LIN {X 0,Y 308.222,Z 305.882,A -85,B 0,C 180,E1 -15823.701,E2 -15823.701} C_VEL
LIN {X 0,Y 306.915,Z 363.331,A -85,B 0,C 180,E1 -15825.712,E2 -15825.712} C_VEL
LIN {X 0,Y 306.575,Z 374.52,A -85,B 0,C 180,E1 -15826.33,E2 -15826.33} C_VEL
LIN {X 0,Y 306.13,Z 386.23,A -85,B 0,C 180,E1 -15827.239,E2 -15827.239} C_VEL
LIN {X 0,Y 305.731,Z 395.85,A -85,B 0,C 180,E1 -15828.233,E2 -15828.233} C_VEL
LIN {X 0,Y 305.222,Z 403.664,A -85,B 0,C 180,E1 -15829.222,E2 -15829.222} C_VEL
LIN {X 0,Y 304.911,Z 411.279,A -85,B 0,C 180,E1 -15830.385,E2 -15830.385} C_VEL
LIN {X 0,Y 304.492,Z 420.077,A -85,B 0,C 180,E1 -15832.044,E2 -15832.044} C_VEL
LIN {X 0,Y 304.105,Z 426.542,A -85,B 0,C 180,E1 -15833.594,E2 -15833.594} C_VEL
LIN {X 0,Y 303.997,Z 432.469,A -85,B 0,C 180,E1 -15835.363,E2 -15835.363} C_VEL
LIN {X 0,Y 303.844,Z 436.01,A -85,B 0,C 180,E1 -15836.689,E2 -15836.689} C_VEL
LIN {X 0,Y 303.696,Z 438.88,A -85,B 0,C 180,E1 -15838.015,E2 -15838.015} C_VEL
LIN {X 0,Y 303.696,Z 442.054,A -85,B 0,C 180,E1 -15840.004,E2 -15840.004} C_VEL
LIN {X 0,Y 303.79,Z 443.417,A -85,B 0,C 180,E1 -15841.33,E2 -15841.33} C_VEL
LIN {X 0,Y 303.999,Z 444.25,A -85,B 0,C 180,E1 -15842.654,E2 -15842.654} C_VEL
LIN {X 0,Y 304.362,Z 444.561,A -85,B 0,C 180,E1 -15843.976,E2 -15843.976} C_VEL
LIN {X 0,Y 304.785,Z 444.334,A -85,B 0,C 180,E1 -15845.296,E2 -15845.296} C_VEL
LIN {X 0,Y 305.137,Z 443.516,A -85,B 0,C 180,E1 -15846.617,E2 -15846.617} C_VEL
LIN {X 0,Y 305.482,Z 442.17,A -85,B 0,C 180,E1 -15847.938,E2 -15847.938} C_VEL
LIN {X 0,Y 306.786,Z 439.095,A -85,B 0,C 180,E1 -15849.913,E2 -15849.913} C_VEL
LIN {X 0,Y 308.158,Z 434.613,A -85,B 0,C 180,E1 -15851.848,E2 -15851.848} C_VEL
LIN {X 0,Y 309.858,Z 428.578,A -85,B 0,C 180,E1 -15853.781,E2 -15853.781} C_VEL
LIN {X 0,Y 311.569,Z 422.164,A -85,B 0,C 180,E1 -15855.373,E2 -15855.373} C_VEL
LIN {X 0,Y 313.433,Z 413.992,A -85,B 0,C 180,E1 -15856.951,E2 -15856.951} C_VEL
LIN {X 0,Y 315.28,Z 404.81,A -85,B 0,C 180,E1 -15858.356,E2 -15858.356} C_VEL
LIN {X 0,Y 317.115,Z 394.594,A -85,B 0,C 180,E1 -15859.589,E2 -15859.589} C_VEL
LIN {X 0,Y 318.559,Z 384.696,A -85,B 0,C 180,E1 -15860.505,E2 -15860.505} C_VEL
LIN {X 0,Y 319.952,Z 372.941,A -85,B 0,C 180,E1 -15861.338,E2 -15861.338} C_VEL
LIN {X 0,Y 321.066,Z 360.035,A -85,B 0,C 180,E1 -15861.94,E2 -15861.94} C_VEL
LIN {X 0,Y 324.472,Z 318.367,A -85,B 0,C 180,E1 -15863.552,E2 -15863.552} C_VEL
LIN {X 0,Y 320.07,Z 308.921,A -85,B 0,C 180,E1 -15864.841,E2 -15864.841} C_VEL
LIN {X 0,Y 315.605,Z 300.854,A -85,B 0,C 180,E1 -15866.21,E2 -15866.21} C_VEL
LIN {X 0,Y 313.092,Z 296.819,A -85,B 0,C 180,E1 -15867.028,E2 -15867.028} C_VEL
LIN {X 0,Y 310.13,Z 292.309,A -85,B 0,C 180,E1 -15868.032,E2 -15868.032} C_VEL
LIN {X 0,Y 307.849,Z 288.757,A -85,B 0,C 180,E1 -15868.912,E2 -15868.912} C_VEL
LIN {X 0,Y 306.286,Z 284.748,A -85,B 0,C 180,E1 -15871.087,E2 -15871.087} C_VEL
LIN {X 0,Y 305.48,Z 282.247,A -85,B 0,C 180,E1 -15872.536,E2 -15872.536} C_VEL
LIN {X 0,Y 305.461,Z 282.248,A -85,B 0,C 180,E1 -15876.745,E2 -15876.745} C_VEL
LIN {X 0,Y 305.42,Z 282.253,A -85,B 0,C 180,E1 -15880.592,E2 -15880.592} C_VEL
LIN {X 0,Y 305.432,Z 282.249,A -85,B 0,C 180,E1 -15883.658,E2 -15883.658} C_VEL
LIN {X 0,Y 305.453,Z 282.246,A -85,B 0,C 180,E1 -15887.419,E2 -15887.419} C_VEL
LIN {X 0,Y 305.469,Z 282.246,A -85,B 0,C 180,E1 -15889.894,E2 -15889.894} C_VEL
LIN {X 0,Y 305.474,Z 282.24,A -85,B 0,C 180,E1 -15893.638,E2 -15893.638} C_VEL
LIN {X 0,Y 305.483,Z 282.361,A -85,B 0,C 180,E1 -15896.831,E2 -15896.831} C_VEL
LIN {X 0,Y 306.911,Z 285.743,A -85,B 0,C 180,E1 -15898.218,E2 -15898.218} C_VEL
LIN {X 0,Y 308.188,Z 287.872,A -85,B 0,C 180,E1 -15899.13,E2 -15899.13} C_VEL
LIN {X 0,Y 311.974,Z 294.665,A -85,B 0,C 180,E1 -15901.475,E2 -15901.475} C_VEL
LIN {X 0,Y 313.574,Z 299.445,A -85,B 0,C 180,E1 -15902.559,E2 -15902.559} C_VEL
LIN {X 0,Y 316.579,Z 307.966,A -85,B 0,C 180,E1 -15903.728,E2 -15903.728} C_VEL
LIN {X 0,Y 319.09,Z 321.708,A -85,B 0,C 180,E1 -15905.03,E2 -15905.03} C_VEL
LIN {X 0,Y 321.279,Z 340.372,A -85,B 0,C 180,E1 -15906.429,E2 -15906.429} C_VEL
LIN {X 0,Y 321.899,Z 352.846,A -85,B 0,C 180,E1 -15907.185,E2 -15907.185} C_VEL
LIN {X 0,Y 318.853,Z 391.341,A -85,B 0,C 180,E1 -15908.715,E2 -15908.715} C_VEL
LIN {X 0,Y 317.251,Z 403.092,A -85,B 0,C 180,E1 -15909.41,E2 -15909.41} C_VEL
LIN {X 0,Y 315.418,Z 414.235,A -85,B 0,C 180,E1 -15910.305,E2 -15910.305} C_VEL
LIN {X 0,Y 313.271,Z 425.528,A -85,B 0,C 180,E1 -15911.525,E2 -15911.525} C_VEL
LIN {X 0,Y 311.637,Z 433.396,A -85,B 0,C 180,E1 -15912.613,E2 -15912.613} C_VEL
LIN {X 0,Y 310.356,Z 439.144,A -85,B 0,C 180,E1 -15913.557,E2 -15913.557} C_VEL
LIN {X 0,Y 308.572,Z 447.09,A -85,B 0,C 180,E1 -15915.153,E2 -15915.153} C_VEL
LIN {X 0,Y 307.019,Z 453.583,A -85,B 0,C 180,E1 -15916.767,E2 -15916.767} C_VEL
LIN {X 0,Y 305.696,Z 459.553,A -85,B 0,C 180,E1 -15918.731,E2 -15918.731} C_VEL
LIN {X 0,Y 304.665,Z 464.003,A -85,B 0,C 180,E1 -15920.707,E2 -15920.707} C_VEL
LIN {X 0,Y 304.18,Z 466.239,A -85,B 0,C 180,E1 -15922.031,E2 -15922.031} C_VEL
LIN {X 0,Y 303.857,Z 467.931,A -85,B 0,C 180,E1 -15923.359,E2 -15923.359} C_VEL
LIN {X 0,Y 303.703,Z 469.072,A -85,B 0,C 180,E1 -15924.689,E2 -15924.689} C_VEL
LIN {X 0,Y 303.705,Z 469.6,A -85,B 0,C 180,E1 -15926.019,E2 -15926.019} C_VEL
LIN {X 0,Y 303.7,Z 469.578,A -85,B 0,C 180,E1 -15927.347,E2 -15927.347} C_VEL
LIN {X 0,Y 303.732,Z 470.856,A -85,B 0,C 180,E1 -15928.674,E2 -15928.674} C_VEL
LIN {X 0,Y 303.767,Z 471.719,A -85,B 0,C 180,E1 -15930,E2 -15930} C_VEL
LIN {X 0,Y 303.675,Z 472.01,A -85,B 0,C 180,E1 -15931.326,E2 -15931.326} C_VEL
LIN {X 0,Y 303.669,Z 471.757,A -85,B 0,C 180,E1 -15932.653,E2 -15932.653} C_VEL
LIN {X 0,Y 303.693,Z 471.045,A -85,B 0,C 180,E1 -15933.981,E2 -15933.981} C_VEL
LIN {X 0,Y 303.741,Z 469.324,A -85,B 0,C 180,E1 -15935.745,E2 -15935.745} C_VEL
LIN {X 0,Y 303.981,Z 467.036,A -85,B 0,C 180,E1 -15937.305,E2 -15937.305} C_VEL
LIN {X 0,Y 304.552,Z 462.968,A -85,B 0,C 180,E1 -15939.296,E2 -15939.296} C_VEL
LIN {X 0,Y 305.469,Z 457.514,A -85,B 0,C 180,E1 -15941.277,E2 -15941.277} C_VEL
LIN {X 0,Y 306.487,Z 451.586,A -85,B 0,C 180,E1 -15942.919,E2 -15942.919} C_VEL
LIN {X 0,Y 307.726,Z 444.1,A -85,B 0,C 180,E1 -15944.55,E2 -15944.55} C_VEL
LIN {X 0,Y 309.047,Z 436.733,A -85,B 0,C 180,E1 -15945.836,E2 -15945.836} C_VEL
LIN {X 0,Y 310.236,Z 428.868,A -85,B 0,C 180,E1 -15946.957,E2 -15946.957} C_VEL
LIN {X 0,Y 311.491,Z 420.567,A -85,B 0,C 180,E1 -15947.903,E2 -15947.903} C_VEL
LIN {X 0,Y 312.707,Z 410.021,A -85,B 0,C 180,E1 -15948.849,E2 -15948.849} C_VEL
LIN {X 0,Y 313.833,Z 398.627,A -85,B 0,C 180,E1 -15949.543,E2 -15949.543} C_VEL
LIN {X 0,Y 314.465,Z 389.052,A -85,B 0,C 180,E1 -15949.934,E2 -15949.934} C_VEL
LIN {X 0,Y 315.324,Z 349.248,A -85,B 0,C 180,E1 -15950.906,E2 -15950.906} C_VEL
LIN {X 0,Y 312.484,Z 330.482,A -85,B 0,C 180,E1 -15951.629,E2 -15951.629} C_VEL
LIN {X 0,Y 308.344,Z 310.347,A -85,B 0,C 180,E1 -15952.538,E2 -15952.538} C_VEL
LIN {X 0,Y 309.432,Z 302.136,A -85,B 0,C 180,E1 -15954.993,E2 -15954.993} C_VEL
LIN {X 0,Y 308.381,Z 295.263,A -85,B 0,C 180,E1 -15957.271,E2 -15957.271} C_VEL
LIN {X 0,Y 306.222,Z 285.499,A -85,B 0,C 180,E1 -15960.707,E2 -15960.707} C_VEL
LIN {X 0,Y 305.446,Z 282.244,A -85,B 0,C 180,E1 -15961.952,E2 -15961.952} C_VEL
LIN {X 0,Y 305.47,Z 282.239,A -85,B 0,C 180,E1 -15965.112,E2 -15965.112} C_VEL
LIN {X 0,Y 305.436,Z 282.251,A -85,B 0,C 180,E1 -15968.521,E2 -15968.521} C_VEL
LIN {X 0,Y 305.449,Z 282.248,A -85,B 0,C 180,E1 -15971.855,E2 -15971.855} C_VEL
LIN {X 0,Y 305.409,Z 282.255,A -85,B 0,C 180,E1 -15975.509,E2 -15975.509} C_VEL
LIN {X 0,Y 305.421,Z 282.251,A -85,B 0,C 180,E1 -15978.136,E2 -15978.136} C_VEL
LIN {X 0,Y 305.45,Z 282.244,A -85,B 0,C 180,E1 -15981.59,E2 -15981.59} C_VEL
LIN {X 0,Y 305.47,Z 282.238,A -85,B 0,C 180,E1 -15984.884,E2 -15984.884} C_VEL
LIN {X 0,Y 305.449,Z 282.242,A -85,B 0,C 180,E1 -15988.356,E2 -15988.356} C_VEL
LIN {X 0,Y 305.493,Z 282.242,A -85,B 0,C 180,E1 -15991.107,E2 -15991.107} C_VEL
LIN {X 0,Y 305.51,Z 282.235,A -85,B 0,C 180,E1 -15994.079,E2 -15994.079} C_VEL
LIN {X 0,Y 305.481,Z 282.234,A -85,B 0,C 180,E1 -15998.398,E2 -15998.398} C_VEL
LIN {X 0,Y 305.548,Z 282.235,A -85,B 0,C 180,E1 -16001.211,E2 -16001.211} C_VEL
LIN {X 0,Y 305.631,Z 282.22,A -85,B 0,C 180,E1 -16005.344,E2 -16005.344} C_VEL
LIN {X 0,Y 305.639,Z 282.21,A -85,B 0,C 180,E1 -16009.396,E2 -16009.396} C_VEL
LIN {X 0,Y 305.8,Z 282.202,A -85,B 0,C 180,E1 -16012.07,E2 -16012.07} C_VEL
LIN {X 0,Y 305.681,Z 282.205,A -85,B 0,C 180,E1 -16014.719,E2 -16014.719} C_VEL
LIN {X 0,Y 305.952,Z 282.176,A -85,B 0,C 180,E1 -16018.68,E2 -16018.68} C_VEL
LIN {X 0,Y 305.951,Z 282.178,A -85,B 0,C 180,E1 -16021.312,E2 -16021.312} C_VEL
LIN {X 0,Y 305.669,Z 282.207,A -85,B 0,C 180,E1 -16025.272,E2 -16025.272} C_VEL
LIN {X 0,Y 305.76,Z 282.209,A -85,B 0,C 180,E1 -16027.922,E2 -16027.922} C_VEL
LIN {X 0,Y 305.594,Z 282.225,A -85,B 0,C 180,E1 -16031.941,E2 -16031.941} C_VEL
LIN {X 0,Y 305.631,Z 282.218,A -85,B 0,C 180,E1 -16035.03,E2 -16035.03} C_VEL
LIN {X 0,Y 305.568,Z 282.23,A -85,B 0,C 180,E1 -16039.44,E2 -16039.44} C_VEL
LIN {X 0,Y 305.48,Z 282.244,A -85,B 0,C 180,E1 -16043.037,E2 -16043.037} C_VEL
LIN {X 0,Y 305.534,Z 282.238,A -85,B 0,C 180,E1 -16046.222,E2 -16046.222} C_VEL
LIN {X 0,Y 305.474,Z 282.244,A -85,B 0,C 180,E1 -16049.043,E2 -16049.043} C_VEL
LIN {X 0,Y 305.426,Z 282.248,A -85,B 0,C 180,E1 -16051.948,E2 -16051.948} C_VEL
LIN {X 0,Y 305.445,Z 282.237,A -85,B 0,C 180,E1 -16055.109,E2 -16055.109} C_VEL
LIN {X 0,Y 305.464,Z 282.25,A -85,B 0,C 180,E1 -16058.532,E2 -16058.532} C_VEL
LIN {X 0,Y 305.5,Z 282.247,A -85,B 0,C 180,E1 -16062.595,E2 -16062.595} C_VEL
LIN {X 0,Y 305.511,Z 282.24,A -85,B 0,C 180,E1 -16066.36,E2 -16066.36} C_VEL
LIN {X 0,Y 305.504,Z 282.301,A -85,B 0,C 180,E1 -16069.07,E2 -16069.07} C_VEL
LIN {X 0,Y 306.197,Z 285.476,A -85,B 0,C 180,E1 -16070.276,E2 -16070.276} C_VEL
LIN {X 0,Y 314.034,Z 303.632,A -85,B 0,C 180,E1 -16071.501,E2 -16071.501} C_VEL
LIN {X 0,Y 315.844,Z 309.078,A -85,B 0,C 180,E1 -16071.805,E2 -16071.805} C_VEL
LIN {X 0,Y 316.318,Z 312.256,A -85,B 0,C 180,E1 -16071.928,E2 -16071.928} C_VEL
LIN {X 0,Y 315.025,Z 362.447,A -85,B 0,C 180,E1 -16073.124,E2 -16073.124} C_VEL
LIN {X 0,Y 314.521,Z 372.658,A -85,B 0,C 180,E1 -16073.558,E2 -16073.558} C_VEL
LIN {X 0,Y 313.622,Z 384.807,A -85,B 0,C 180,E1 -16074.364,E2 -16074.364} C_VEL
LIN {X 0,Y 312.594,Z 394.073,A -85,B 0,C 180,E1 -16075.215,E2 -16075.215} C_VEL
LIN {X 0,Y 311.639,Z 402.117,A -85,B 0,C 180,E1 -16076.158,E2 -16076.158} C_VEL
LIN {X 0,Y 310.511,Z 409.965,A -85,B 0,C 180,E1 -16077.291,E2 -16077.291} C_VEL
LIN {X 0,Y 309.347,Z 416.815,A -85,B 0,C 180,E1 -16078.498,E2 -16078.498} C_VEL
LIN {X 0,Y 308.024,Z 424.176,A -85,B 0,C 180,E1 -16080.102,E2 -16080.102} C_VEL
LIN {X 0,Y 306.792,Z 430.833,A -85,B 0,C 180,E1 -16081.991,E2 -16081.991} C_VEL
LIN {X 0,Y 305.862,Z 435.31,A -85,B 0,C 180,E1 -16083.64,E2 -16083.64} C_VEL
LIN {X 0,Y 305.059,Z 439.119,A -85,B 0,C 180,E1 -16085.501,E2 -16085.501} C_VEL
LIN {X 0,Y 304.433,Z 441.868,A -85,B 0,C 180,E1 -16087.415,E2 -16087.415} C_VEL
LIN {X 0,Y 304.202,Z 442.815,A -85,B 0,C 180,E1 -16088.306,E2 -16088.306} C_VEL
LIN {X 0,Y 303.9,Z 443.783,A -85,B 0,C 180,E1 -16089.703,E2 -16089.703} C_VEL
LIN {X 0,Y 303.654,Z 444.181,A -85,B 0,C 180,E1 -16091.591,E2 -16091.591} C_VEL
LIN {X 0,Y 303.571,Z 443.264,A -85,B 0,C 180,E1 -16093.871,E2 -16093.871} C_VEL
LIN {X 0,Y 303.662,Z 442.055,A -85,B 0,C 180,E1 -16095.251,E2 -16095.251} C_VEL
LIN {X 0,Y 303.816,Z 440.306,A -85,B 0,C 180,E1 -16096.625,E2 -16096.625} C_VEL
LIN {X 0,Y 304.15,Z 436.443,A -85,B 0,C 180,E1 -16098.673,E2 -16098.673} C_VEL
LIN {X 0,Y 304.596,Z 431.173,A -85,B 0,C 180,E1 -16100.706,E2 -16100.706} C_VEL
LIN {X 0,Y 305.064,Z 425.345,A -85,B 0,C 180,E1 -16102.436,E2 -16102.436} C_VEL
LIN {X 0,Y 305.742,Z 418.331,A -85,B 0,C 180,E1 -16104.063,E2 -16104.063} C_VEL
LIN {X 0,Y 306.469,Z 410.103,A -85,B 0,C 180,E1 -16105.561,E2 -16105.561} C_VEL
LIN {X 0,Y 307.174,Z 402.221,A -85,B 0,C 180,E1 -16106.721,E2 -16106.721} C_VEL
LIN {X 0,Y 307.818,Z 393.913,A -85,B 0,C 180,E1 -16107.71,E2 -16107.71} C_VEL
LIN {X 0,Y 308.409,Z 385.228,A -85,B 0,C 180,E1 -16108.531,E2 -16108.531} C_VEL
LIN {X 0,Y 309,Z 373.68,A -85,B 0,C 180,E1 -16109.349,E2 -16109.349} C_VEL
LIN {X 0,Y 309.302,Z 362.42,A -85,B 0,C 180,E1 -16109.854,E2 -16109.854} C_VEL
LIN {X 0,Y 309.849,Z 331.975,A -85,B 0,C 180,E1 -16110.602,E2 -16110.602} C_VEL
LIN {X 0,Y 310.282,Z 307.413,A -85,B 0,C 180,E1 -16111.166,E2 -16111.166} C_VEL
LIN {X 0,Y 306.839,Z 286.854,A -85,B 0,C 180,E1 -16111.821,E2 -16111.821} C_VEL
LIN {X 0,Y 306.326,Z 284.637,A -85,B 0,C 180,E1 -16111.927,E2 -16111.927} C_VEL
LIN {X 0,Y 305.818,Z 282.207,A -85,B 0,C 180,E1 -16112.799,E2 -16112.799} C_VEL
LIN {X 0,Y 305.808,Z 282.203,A -85,B 0,C 180,E1 -16116.599,E2 -16116.599} C_VEL
LIN {X 0,Y 305.671,Z 282.224,A -85,B 0,C 180,E1 -16119.262,E2 -16119.262} C_VEL
LIN {X 0,Y 305.555,Z 282.238,A -85,B 0,C 180,E1 -16123.298,E2 -16123.298} C_VEL
LIN {X 0,Y 305.528,Z 282.237,A -85,B 0,C 180,E1 -16126.024,E2 -16126.024} C_VEL
LIN {X 0,Y 305.546,Z 282.239,A -85,B 0,C 180,E1 -16129.447,E2 -16129.447} C_VEL
LIN {X 0,Y 305.457,Z 282.248,A -85,B 0,C 180,E1 -16133.042,E2 -16133.042} C_VEL
LIN {X 0,Y 305.44,Z 282.248,A -85,B 0,C 180,E1 -16136.2,E2 -16136.2} C_VEL
LIN {X 0,Y 305.42,Z 282.252,A -85,B 0,C 180,E1 -16139.037,E2 -16139.037} C_VEL
LIN {X 0,Y 305.409,Z 282.252,A -85,B 0,C 180,E1 -16141.957,E2 -16141.957} C_VEL
LIN {X 0,Y 305.436,Z 282.249,A -85,B 0,C 180,E1 -16145.117,E2 -16145.117} C_VEL
LIN {X 0,Y 305.409,Z 282.25,A -85,B 0,C 180,E1 -16148.529,E2 -16148.529} C_VEL
LIN {X 0,Y 305.413,Z 282.25,A -85,B 0,C 180,E1 -16152.586,E2 -16152.586} C_VEL
LIN {X 0,Y 305.405,Z 282.252,A -85,B 0,C 180,E1 -16156.349,E2 -16156.349} C_VEL
LIN {X 0,Y 305.44,Z 282.251,A -85,B 0,C 180,E1 -16159.897,E2 -16159.897} C_VEL
LIN {X 0,Y 305.465,Z 282.248,A -85,B 0,C 180,E1 -16163.636,E2 -16163.636} C_VEL
LIN {X 0,Y 305.45,Z 282.246,A -85,B 0,C 180,E1 -16166.488,E2 -16166.488} C_VEL
LIN {X 0,Y 305.417,Z 282.252,A -85,B 0,C 180,E1 -16169.592,E2 -16169.592} C_VEL
LIN {X 0,Y 305.461,Z 282.245,A -85,B 0,C 180,E1 -16171.143,E2 -16171.143} C_VEL
LIN {X 0,Y 304.749,Z 282.336,A -85,B 0,C 180,E1 -16172.244,E2 -16172.244} C_VEL
LIN {X 0,Y 301.911,Z 282.691,A -85,B 0,C 180,E1 -16174.038,E2 -16174.038} C_VEL
LIN {X 0,Y 299.528,Z 282.985,A -85,B 0,C 180,E1 -16175.493,E2 -16175.493} C_VEL
LIN {X 0,Y 298.495,Z 283.111,A -85,B 0,C 180,E1 -16176.619,E2 -16176.619} C_VEL
LIN {X 0,Y 298.403,Z 283.121,A -85,B 0,C 180,E1 -16177,E2 -16177} C_VEL
LIN {X 0,Y 298.54,Z 283.097,A -85,B 0,C 180,E1 -16180.762,E2 -16180.762} C_VEL
LIN {X 0,Y 298.622,Z 283.234,A -85,B 0,C 180,E1 -16182.676,E2 -16182.676} C_VEL
LIN {X 0,Y 300.215,Z 298.823,A -85,B 0,C 180,E1 -16183.302,E2 -16183.302} C_VEL
LIN {X 0,Y 301.125,Z 306.72,A -85,B 0,C 180,E1 -16183.6,E2 -16183.6} C_VEL
LIN {X 0,Y 299.839,Z 362.846,A -85,B 0,C 180,E1 -16185.628,E2 -16185.628} C_VEL
LIN {X 0,Y 299.492,Z 374.119,A -85,B 0,C 180,E1 -16186.26,E2 -16186.26} C_VEL
LIN {X 0,Y 299.077,Z 385.094,A -85,B 0,C 180,E1 -16187.105,E2 -16187.105} C_VEL
LIN {X 0,Y 298.707,Z 394.969,A -85,B 0,C 180,E1 -16188.124,E2 -16188.124} C_VEL
LIN {X 0,Y 298.107,Z 404.115,A -85,B 0,C 180,E1 -16189.305,E2 -16189.305} C_VEL
LIN {X 0,Y 297.79,Z 411.698,A -85,B 0,C 180,E1 -16190.496,E2 -16190.496} C_VEL
LIN {X 0,Y 297.377,Z 420.49,A -85,B 0,C 180,E1 -16192.195,E2 -16192.195} C_VEL
LIN {X 0,Y 297.021,Z 426.353,A -85,B 0,C 180,E1 -16193.613,E2 -16193.613} C_VEL
LIN {X 0,Y 296.921,Z 431.88,A -85,B 0,C 180,E1 -16195.253,E2 -16195.253} C_VEL
LIN {X 0,Y 296.779,Z 435.618,A -85,B 0,C 180,E1 -16196.61,E2 -16196.61} C_VEL
LIN {X 0,Y 296.594,Z 439.93,A -85,B 0,C 180,E1 -16198.647,E2 -16198.647} C_VEL
LIN {X 0,Y 296.607,Z 441.999,A -85,B 0,C 180,E1 -16200.004,E2 -16200.004} C_VEL
LIN {X 0,Y 296.703,Z 443.52,A -85,B 0,C 180,E1 -16201.362,E2 -16201.362} C_VEL
LIN {X 0,Y 296.92,Z 444.52,A -85,B 0,C 180,E1 -16202.718,E2 -16202.718} C_VEL
LIN {X 0,Y 297.293,Z 444.97,A -85,B 0,C 180,E1 -16204.071,E2 -16204.071} C_VEL
LIN {X 0,Y 297.727,Z 444.813,A -85,B 0,C 180,E1 -16205.422,E2 -16205.422} C_VEL
LIN {X 0,Y 298.1,Z 444.132,A -85,B 0,C 180,E1 -16206.774,E2 -16206.774} C_VEL
LIN {X 0,Y 298.509,Z 442.948,A -85,B 0,C 180,E1 -16208.125,E2 -16208.125} C_VEL
LIN {X 0,Y 299.91,Z 440.008,A -85,B 0,C 180,E1 -16210.191,E2 -16210.191} C_VEL
LIN {X 0,Y 301.345,Z 435.986,A -85,B 0,C 180,E1 -16212.12,E2 -16212.12} C_VEL
LIN {X 0,Y 303.141,Z 430.181,A -85,B 0,C 180,E1 -16214.093,E2 -16214.093} C_VEL
LIN {X 0,Y 304.93,Z 423.995,A -85,B 0,C 180,E1 -16215.716,E2 -16215.716} C_VEL
LIN {X 0,Y 306.945,Z 416.421,A -85,B 0,C 180,E1 -16217.321,E2 -16217.321} C_VEL
LIN {X 0,Y 308.881,Z 407.739,A -85,B 0,C 180,E1 -16218.751,E2 -16218.751} C_VEL
LIN {X 0,Y 310.546,Z 399.443,A -85,B 0,C 180,E1 -16219.848,E2 -16219.848} C_VEL
LIN {X 0,Y 312.291,Z 389.225,A -85,B 0,C 180,E1 -16220.936,E2 -16220.936} C_VEL
LIN {X 0,Y 313.868,Z 377.612,A -85,B 0,C 180,E1 -16221.859,E2 -16221.859} C_VEL
LIN {X 0,Y 315.22,Z 365.425,A -85,B 0,C 180,E1 -16222.555,E2 -16222.555} C_VEL
LIN {X 0,Y 319.095,Z 321.02,A -85,B 0,C 180,E1 -16224.323,E2 -16224.323} C_VEL
LIN {X 0,Y 315.052,Z 312.283,A -85,B 0,C 180,E1 -16225.618,E2 -16225.618} C_VEL
LIN {X 0,Y 311.131,Z 305.071,A -85,B 0,C 180,E1 -16226.921,E2 -16226.921} C_VEL
LIN {X 0,Y 306.842,Z 298.193,A -85,B 0,C 180,E1 -16228.439,E2 -16228.439} C_VEL
LIN {X 0,Y 303.696,Z 293.645,A -85,B 0,C 180,E1 -16229.656,E2 -16229.656} C_VEL
LIN {X 0,Y 300.828,Z 289.417,A -85,B 0,C 180,E1 -16230.932,E2 -16230.932} C_VEL
LIN {X 0,Y 299.893,Z 286.637,A -85,B 0,C 180,E1 -16232.62,E2 -16232.62} C_VEL
LIN {X 0,Y 298.432,Z 283.124,A -85,B 0,C 180,E1 -16235.241,E2 -16235.241} C_VEL
LIN {X 0,Y 298.395,Z 283.128,A -85,B 0,C 180,E1 -16238.991,E2 -16238.991} C_VEL
LIN {X 0,Y 298.381,Z 283.128,A -85,B 0,C 180,E1 -16243.099,E2 -16243.099} C_VEL
LIN {X 0,Y 298.386,Z 283.128,A -85,B 0,C 180,E1 -16246.917,E2 -16246.917} C_VEL
LIN {X 0,Y 298.406,Z 283.127,A -85,B 0,C 180,E1 -16251.01,E2 -16251.01} C_VEL
LIN {X 0,Y 298.456,Z 283.255,A -85,B 0,C 180,E1 -16254.039,E2 -16254.039} C_VEL
LIN {X 0,Y 299.715,Z 286.364,A -85,B 0,C 180,E1 -16255.752,E2 -16255.752} C_VEL
LIN {X 0,Y 300.758,Z 287.513,A -85,B 0,C 180,E1 -16256.48,E2 -16256.48} C_VEL
LIN {X 0,Y 301.778,Z 290.151,A -85,B 0,C 180,E1 -16257.612,E2 -16257.612} C_VEL
LIN {X 0,Y 304.349,Z 294.686,A -85,B 0,C 180,E1 -16259.468,E2 -16259.468} C_VEL
LIN {X 0,Y 306.484,Z 298.591,A -85,B 0,C 180,E1 -16260.785,E2 -16260.785} C_VEL
LIN {X 0,Y 308.269,Z 301.368,A -85,B 0,C 180,E1 -16261.447,E2 -16261.447} C_VEL
LIN {X 0,Y 310.441,Z 306.807,A -85,B 0,C 180,E1 -16262.333,E2 -16262.333} C_VEL
LIN {X 0,Y 312.113,Z 312.313,A -85,B 0,C 180,E1 -16263.072,E2 -16263.072} C_VEL
LIN {X 0,Y 314.172,Z 324.681,A -85,B 0,C 180,E1 -16264.268,E2 -16264.268} C_VEL
LIN {X 0,Y 315.937,Z 341.809,A -85,B 0,C 180,E1 -16265.611,E2 -16265.611} C_VEL
LIN {X 0,Y 316.494,Z 353.234,A -85,B 0,C 180,E1 -16266.34,E2 -16266.34} C_VEL
LIN {X 0,Y 313.237,Z 391.388,A -85,B 0,C 180,E1 -16267.925,E2 -16267.925} C_VEL
LIN {X 0,Y 311.475,Z 403.471,A -85,B 0,C 180,E1 -16268.664,E2 -16268.664} C_VEL
LIN {X 0,Y 309.544,Z 414.385,A -85,B 0,C 180,E1 -16269.569,E2 -16269.569} C_VEL
LIN {X 0,Y 307.259,Z 425.398,A -85,B 0,C 180,E1 -16270.804,E2 -16270.804} C_VEL
LIN {X 0,Y 305.234,Z 434.196,A -85,B 0,C 180,E1 -16272.063,E2 -16272.063} C_VEL
LIN {X 0,Y 303.28,Z 442.361,A -85,B 0,C 180,E1 -16273.508,E2 -16273.508} C_VEL
LIN {X 0,Y 301.481,Z 449.559,A -85,B 0,C 180,E1 -16275.142,E2 -16275.142} C_VEL
LIN {X 0,Y 299.904,Z 455.347,A -85,B 0,C 180,E1 -16276.792,E2 -16276.792} C_VEL
LIN {X 0,Y 298.739,Z 459.998,A -85,B 0,C 180,E1 -16278.465,E2 -16278.465} C_VEL
LIN {X 0,Y 297.968,Z 462.986,A -85,B 0,C 180,E1 -16279.811,E2 -16279.811} C_VEL
LIN {X 0,Y 297.134,Z 466.307,A -85,B 0,C 180,E1 -16281.841,E2 -16281.841} C_VEL
LIN {X 0,Y 296.642,Z 468.726,A -85,B 0,C 180,E1 -16284.324,E2 -16284.324} C_VEL
LIN {X 0,Y 296.619,Z 469.295,A -85,B 0,C 180,E1 -16285.924,E2 -16285.924} C_VEL
LIN {X 0,Y 296.622,Z 469.141,A -85,B 0,C 180,E1 -16287.284,E2 -16287.284} C_VEL
LIN {X 0,Y 296.643,Z 470.452,A -85,B 0,C 180,E1 -16288.642,E2 -16288.642} C_VEL
LIN {X 0,Y 296.676,Z 471.354,A -85,B 0,C 180,E1 -16290,E2 -16290} C_VEL
LIN {X 0,Y 296.589,Z 471.656,A -85,B 0,C 180,E1 -16291.358,E2 -16291.358} C_VEL
LIN {X 0,Y 296.593,Z 471.455,A -85,B 0,C 180,E1 -16292.716,E2 -16292.716} C_VEL
LIN {X 0,Y 296.608,Z 470.793,A -85,B 0,C 180,E1 -16294.076,E2 -16294.076} C_VEL
LIN {X 0,Y 296.642,Z 469.377,A -85,B 0,C 180,E1 -16295.675,E2 -16295.675} C_VEL
LIN {X 0,Y 296.912,Z 466.891,A -85,B 0,C 180,E1 -16297.48,E2 -16297.48} C_VEL
LIN {X 0,Y 297.538,Z 462.882,A -85,B 0,C 180,E1 -16299.517,E2 -16299.517} C_VEL
LIN {X 0,Y 298.133,Z 459.427,A -85,B 0,C 180,E1 -16300.87,E2 -16300.87} C_VEL
LIN {X 0,Y 299.131,Z 454.092,A -85,B 0,C 180,E1 -16302.552,E2 -16302.552} C_VEL
LIN {X 0,Y 300.084,Z 448.872,A -85,B 0,C 180,E1 -16303.89,E2 -16303.89} C_VEL
LIN {X 0,Y 301.196,Z 442.613,A -85,B 0,C 180,E1 -16305.218,E2 -16305.218} C_VEL
LIN {X 0,Y 302.622,Z 435.016,A -85,B 0,C 180,E1 -16306.528,E2 -16306.528} C_VEL
LIN {X 0,Y 304.156,Z 425.608,A -85,B 0,C 180,E1 -16307.828,E2 -16307.828} C_VEL
LIN {X 0,Y 305.375,Z 416.504,A -85,B 0,C 180,E1 -16308.796,E2 -16308.796} C_VEL
LIN {X 0,Y 306.524,Z 406.574,A -85,B 0,C 180,E1 -16309.592,E2 -16309.592} C_VEL
LIN {X 0,Y 307.485,Z 396.968,A -85,B 0,C 180,E1 -16310.147,E2 -16310.147} C_VEL
LIN {X 0,Y 308.054,Z 388.085,A -85,B 0,C 180,E1 -16310.504,E2 -16310.504} C_VEL
LIN {X 0,Y 308.893,Z 349.93,A -85,B 0,C 180,E1 -16311.454,E2 -16311.454} C_VEL
LIN {X 0,Y 306.203,Z 332.08,A -85,B 0,C 180,E1 -16312.168,E2 -16312.168} C_VEL
LIN {X 0,Y 302.117,Z 312.34,A -85,B 0,C 180,E1 -16313.087,E2 -16313.087} C_VEL
LIN {X 0,Y 301.638,Z 309.982,A -85,B 0,C 180,E1 -16313.202,E2 -16313.202} C_VEL
LIN {X 0,Y 302.502,Z 304.017,A -85,B 0,C 180,E1 -16315.025,E2 -16315.025} C_VEL
LIN {X 0,Y 301.757,Z 298.21,A -85,B 0,C 180,E1 -16316.978,E2 -16316.978} C_VEL
LIN {X 0,Y 299.753,Z 288.706,A -85,B 0,C 180,E1 -16320.376,E2 -16320.376} C_VEL
LIN {X 0,Y 298.401,Z 283.12,A -85,B 0,C 180,E1 -16322.515,E2 -16322.515} C_VEL
LIN {X 0,Y 298.413,Z 283.115,A -85,B 0,C 180,E1 -16326.07,E2 -16326.07} C_VEL
LIN {X 0,Y 298.406,Z 283.126,A -85,B 0,C 180,E1 -16329.486,E2 -16329.486} C_VEL
LIN {X 0,Y 298.409,Z 283.128,A -85,B 0,C 180,E1 -16333.101,E2 -16333.101} C_VEL
LIN {X 0,Y 298.38,Z 283.127,A -85,B 0,C 180,E1 -16336.913,E2 -16336.913} C_VEL
LIN {X 0,Y 298.359,Z 283.125,A -85,B 0,C 180,E1 -16341.017,E2 -16341.017} C_VEL
LIN {X 0,Y 298.412,Z 283.12,A -85,B 0,C 180,E1 -16343.926,E2 -16343.926} C_VEL
LIN {X 0,Y 298.4,Z 283.127,A -85,B 0,C 180,E1 -16347.197,E2 -16347.197} C_VEL
LIN {X 0,Y 298.415,Z 283.123,A -85,B 0,C 180,E1 -16350.62,E2 -16350.62} C_VEL
LIN {X 0,Y 298.454,Z 283.116,A -85,B 0,C 180,E1 -16354.917,E2 -16354.917} C_VEL
LIN {X 0,Y 298.435,Z 283.112,A -85,B 0,C 180,E1 -16359.31,E2 -16359.31} C_VEL
LIN {X 0,Y 298.509,Z 283.108,A -85,B 0,C 180,E1 -16362.174,E2 -16362.174} C_VEL
LIN {X 0,Y 298.59,Z 283.095,A -85,B 0,C 180,E1 -16364.991,E2 -16364.991} C_VEL
LIN {X 0,Y 298.595,Z 283.086,A -85,B 0,C 180,E1 -16369.143,E2 -16369.143} C_VEL
LIN {X 0,Y 298.744,Z 283.082,A -85,B 0,C 180,E1 -16371.881,E2 -16371.881} C_VEL
LIN {X 0,Y 298.653,Z 283.08,A -85,B 0,C 180,E1 -16374.595,E2 -16374.595} C_VEL
LIN {X 0,Y 298.919,Z 283.052,A -85,B 0,C 180,E1 -16378.648,E2 -16378.648} C_VEL
LIN {X 0,Y 298.918,Z 283.054,A -85,B 0,C 180,E1 -16381.343,E2 -16381.343} C_VEL
LIN {X 0,Y 298.638,Z 283.082,A -85,B 0,C 180,E1 -16385.397,E2 -16385.397} C_VEL
LIN {X 0,Y 298.709,Z 283.089,A -85,B 0,C 180,E1 -16388.111,E2 -16388.111} C_VEL
LIN {X 0,Y 298.545,Z 283.106,A -85,B 0,C 180,E1 -16392.227,E2 -16392.227} C_VEL
LIN {X 0,Y 298.599,Z 283.094,A -85,B 0,C 180,E1 -16395.204,E2 -16395.204} C_VEL
LIN {X 0,Y 298.53,Z 283.107,A -85,B 0,C 180,E1 -16399.238,E2 -16399.238} C_VEL
LIN {X 0,Y 298.446,Z 283.119,A -85,B 0,C 180,E1 -16403.593,E2 -16403.593} C_VEL
LIN {X 0,Y 298.477,Z 283.12,A -85,B 0,C 180,E1 -16406.57,E2 -16406.57} C_VEL
LIN {X 0,Y 298.402,Z 283.126,A -85,B 0,C 180,E1 -16409.637,E2 -16409.637} C_VEL
LIN {X 0,Y 298.378,Z 283.131,A -85,B 0,C 180,E1 -16412.796,E2 -16412.796} C_VEL
LIN {X 0,Y 298.434,Z 283.112,A -85,B 0,C 180,E1 -16416.805,E2 -16416.805} C_VEL
LIN {X 0,Y 298.433,Z 283.116,A -85,B 0,C 180,E1 -16421.098,E2 -16421.098} C_VEL
LIN {X 0,Y 298.467,Z 283.117,A -85,B 0,C 180,E1 -16425.057,E2 -16425.057} C_VEL
LIN {X 0,Y 298.454,Z 283.237,A -85,B 0,C 180,E1 -16428.526,E2 -16428.526} C_VEL
LIN {X 0,Y 299.138,Z 286.093,A -85,B 0,C 180,E1 -16429.575,E2 -16429.575} C_VEL
LIN {X 0,Y 307.167,Z 304.088,A -85,B 0,C 180,E1 -16430.866,E2 -16430.866} C_VEL
LIN {X 0,Y 309.787,Z 311.601,A -85,B 0,C 180,E1 -16431.312,E2 -16431.312} C_VEL
LIN {X 0,Y 309.772,Z 320.508,A -85,B 0,C 180,E1 -16431.542,E2 -16431.542} C_VEL
LIN {X 0,Y 308.592,Z 363.013,A -85,B 0,C 180,E1 -16432.582,E2 -16432.582} C_VEL
LIN {X 0,Y 308.038,Z 373.9,A -85,B 0,C 180,E1 -16433.064,E2 -16433.064} C_VEL
LIN {X 0,Y 307.068,Z 385.718,A -85,B 0,C 180,E1 -16433.889,E2 -16433.889} C_VEL
LIN {X 0,Y 305.993,Z 394.859,A -85,B 0,C 180,E1 -16434.756,E2 -16434.756} C_VEL
LIN {X 0,Y 305.087,Z 402.233,A -85,B 0,C 180,E1 -16435.64,E2 -16435.64} C_VEL
LIN {X 0,Y 303.998,Z 409.511,A -85,B 0,C 180,E1 -16436.697,E2 -16436.697} C_VEL
LIN {X 0,Y 302.917,Z 415.584,A -85,B 0,C 180,E1 -16437.75,E2 -16437.75} C_VEL
LIN {X 0,Y 301.663,Z 422.283,A -85,B 0,C 180,E1 -16439.167,E2 -16439.167} C_VEL
LIN {X 0,Y 300.567,Z 427.781,A -85,B 0,C 180,E1 -16440.592,E2 -16440.592} C_VEL
LIN {X 0,Y 299.665,Z 432.299,A -85,B 0,C 180,E1 -16442.027,E2 -16442.027} C_VEL
LIN {X 0,Y 298.859,Z 435.978,A -85,B 0,C 180,E1 -16443.461,E2 -16443.461} C_VEL
LIN {X 0,Y 297.917,Z 440.127,A -85,B 0,C 180,E1 -16445.617,E2 -16445.617} C_VEL
LIN {X 0,Y 297.245,Z 442.887,A -85,B 0,C 180,E1 -16447.772,E2 -16447.772} C_VEL
LIN {X 0,Y 296.897,Z 443.914,A -85,B 0,C 180,E1 -16449.202,E2 -16449.202} C_VEL
LIN {X 0,Y 296.58,Z 444.518,A -85,B 0,C 180,E1 -16451.398,E2 -16451.398} C_VEL
LIN {X 0,Y 296.468,Z 443.817,A -85,B 0,C 180,E1 -16453.473,E2 -16453.473} C_VEL
LIN {X 0,Y 296.544,Z 442.743,A -85,B 0,C 180,E1 -16454.889,E2 -16454.889} C_VEL
LIN {X 0,Y 296.779,Z 439.963,A -85,B 0,C 180,E1 -16456.999,E2 -16456.999} C_VEL
LIN {X 0,Y 297.118,Z 435.886,A -85,B 0,C 180,E1 -16459.092,E2 -16459.092} C_VEL
LIN {X 0,Y 297.441,Z 432.347,A -85,B 0,C 180,E1 -16460.48,E2 -16460.48} C_VEL
LIN {X 0,Y 297.934,Z 427.054,A -85,B 0,C 180,E1 -16462.151,E2 -16462.151} C_VEL
LIN {X 0,Y 298.43,Z 421.468,A -85,B 0,C 180,E1 -16463.578,E2 -16463.578} C_VEL
LIN {X 0,Y 299.244,Z 413.193,A -85,B 0,C 180,E1 -16465.285,E2 -16465.285} C_VEL
LIN {X 0,Y 300.016,Z 404.694,A -85,B 0,C 180,E1 -16466.643,E2 -16466.643} C_VEL
LIN {X 0,Y 300.673,Z 396.852,A -85,B 0,C 180,E1 -16467.656,E2 -16467.656} C_VEL
LIN {X 0,Y 301.262,Z 388.813,A -85,B 0,C 180,E1 -16468.496,E2 -16468.496} C_VEL
LIN {X 0,Y 301.759,Z 379.587,A -85,B 0,C 180,E1 -16469.25,E2 -16469.25} C_VEL
LIN {X 0,Y 302.194,Z 370.178,A -85,B 0,C 180,E1 -16469.817,E2 -16469.817} C_VEL
LIN {X 0,Y 302.438,Z 360.586,A -85,B 0,C 180,E1 -16470.208,E2 -16470.208} C_VEL
LIN {X 0,Y 303.374,Z 308.078,A -85,B 0,C 180,E1 -16471.473,E2 -16471.473} C_VEL
LIN {X 0,Y 300.128,Z 288.589,A -85,B 0,C 180,E1 -16472.111,E2 -16472.111} C_VEL
LIN {X 0,Y 299.154,Z 284.972,A -85,B 0,C 180,E1 -16472.273,E2 -16472.273} C_VEL
LIN {X 0,Y 298.705,Z 283.094,A -85,B 0,C 180,E1 -16473.035,E2 -16473.035} C_VEL
LIN {X 0,Y 298.753,Z 283.083,A -85,B 0,C 180,E1 -16476.755,E2 -16476.755} C_VEL
LIN {X 0,Y 298.602,Z 283.103,A -85,B 0,C 180,E1 -16479.483,E2 -16479.483} C_VEL
LIN {X 0,Y 298.516,Z 283.113,A -85,B 0,C 180,E1 -16483.617,E2 -16483.617} C_VEL
LIN {X 0,Y 298.496,Z 283.112,A -85,B 0,C 180,E1 -16486.412,E2 -16486.412} C_VEL
LIN {X 0,Y 298.481,Z 283.117,A -85,B 0,C 180,E1 -16489.657,E2 -16489.657} C_VEL
LIN {X 0,Y 298.394,Z 283.129,A -85,B 0,C 180,E1 -16493.603,E2 -16493.603} C_VEL
LIN {X 0,Y 298.379,Z 283.127,A -85,B 0,C 180,E1 -16496.585,E2 -16496.585} C_VEL
LIN {X 0,Y 298.365,Z 283.132,A -85,B 0,C 180,E1 -16499.647,E2 -16499.647} C_VEL
LIN {X 0,Y 298.366,Z 283.127,A -85,B 0,C 180,E1 -16502.804,E2 -16502.804} C_VEL
LIN {X 0,Y 298.401,Z 283.124,A -85,B 0,C 180,E1 -16506.806,E2 -16506.806} C_VEL
LIN {X 0,Y 298.35,Z 283.134,A -85,B 0,C 180,E1 -16509.496,E2 -16509.496} C_VEL
LIN {X 0,Y 298.348,Z 283.131,A -85,B 0,C 180,E1 -16513.102,E2 -16513.102} C_VEL
LIN {X 0,Y 298.384,Z 283.126,A -85,B 0,C 180,E1 -16516.925,E2 -16516.925} C_VEL
LIN {X 0,Y 298.397,Z 283.124,A -85,B 0,C 180,E1 -16521.008,E2 -16521.008} C_VEL
LIN {X 0,Y 298.403,Z 283.129,A -85,B 0,C 180,E1 -16523.935,E2 -16523.935} C_VEL
LIN {X 0,Y 298.374,Z 283.132,A -85,B 0,C 180,E1 -16527.991,E2 -16527.991} C_VEL
LIN {X 0,Y 298.402,Z 283.129,A -85,B 0,C 180,E1 -16531.904,E2 -16531.904} C_VEL
LIN {X 0,Y 298.434,Z 283.119,A -85,B 0,C 180,E1 -16534.925,E2 -16534.925} C_VEL
LIN {X 0,Y 298.403,Z 283.121,A -85,B 0,C 180,E1 -16537,E2 -16537} C_VEL
LIN {X 0,Y 297.717,Z 283.209,A -85,B 0,C 180,E1 -16537.75,E2 -16537.75} C_VEL
LIN {X 0,Y 294.899,Z 283.562,A -85,B 0,C 180,E1 -16538.929,E2 -16538.929} C_VEL
LIN {X 0,Y 292.099,Z 283.909,A -85,B 0,C 180,E1 -16540.129,E2 -16540.129} C_VEL
LIN {X 0,Y 291.467,Z 283.976,A -85,B 0,C 180,E1 -16540.904,E2 -16540.904} C_VEL
LIN {X 0,Y 291.594,Z 283.951,A -85,B 0,C 180,E1 -16542.562,E2 -16542.562} C_VEL
LIN {X 0,Y 293.505,Z 301.908,A -85,B 0,C 180,E1 -16543.297,E2 -16543.297} C_VEL
LIN {X 0,Y 294.081,Z 306.493,A -85,B 0,C 180,E1 -16543.477,E2 -16543.477} C_VEL
LIN {X 0,Y 292.744,Z 363.503,A -85,B 0,C 180,E1 -16545.627,E2 -16545.627} C_VEL
LIN {X 0,Y 292.386,Z 374.659,A -85,B 0,C 180,E1 -16546.274,E2 -16546.274} C_VEL
LIN {X 0,Y 291.982,Z 385.57,A -85,B 0,C 180,E1 -16547.14,E2 -16547.14} C_VEL
LIN {X 0,Y 291.567,Z 395.394,A -85,B 0,C 180,E1 -16548.182,E2 -16548.182} C_VEL
LIN {X 0,Y 291.042,Z 404.557,A -85,B 0,C 180,E1 -16549.395,E2 -16549.395} C_VEL
LIN {X 0,Y 290.54,Z 414.111,A -85,B 0,C 180,E1 -16550.959,E2 -16550.959} C_VEL
LIN {X 0,Y 290.175,Z 422.363,A -85,B 0,C 180,E1 -16552.7,E2 -16552.7} C_VEL
LIN {X 0,Y 289.867,Z 427.547,A -85,B 0,C 180,E1 -16554.026,E2 -16554.026} C_VEL
LIN {X 0,Y 289.816,Z 432.271,A -85,B 0,C 180,E1 -16555.484,E2 -16555.484} C_VEL
LIN {X 0,Y 289.617,Z 436.792,A -85,B 0,C 180,E1 -16557.223,E2 -16557.223} C_VEL
LIN {X 0,Y 289.495,Z 440.907,A -85,B 0,C 180,E1 -16559.309,E2 -16559.309} C_VEL
LIN {X 0,Y 289.619,Z 443.611,A -85,B 0,C 180,E1 -16561.395,E2 -16561.395} C_VEL
LIN {X 0,Y 289.844,Z 444.742,A -85,B 0,C 180,E1 -16562.784,E2 -16562.784} C_VEL
LIN {X 0,Y 290.227,Z 445.268,A -85,B 0,C 180,E1 -16564.17,E2 -16564.17} C_VEL
LIN {X 0,Y 290.672,Z 445.261,A -85,B 0,C 180,E1 -16565.554,E2 -16565.554} C_VEL
LIN {X 0,Y 291.071,Z 444.768,A -85,B 0,C 180,E1 -16566.938,E2 -16566.938} C_VEL
LIN {X 0,Y 291.54,Z 443.783,A -85,B 0,C 180,E1 -16568.321,E2 -16568.321} C_VEL
LIN {X 0,Y 292.576,Z 442.203,A -85,B 0,C 180,E1 -16569.684,E2 -16569.684} C_VEL
LIN {X 0,Y 293.976,Z 438.679,A -85,B 0,C 180,E1 -16571.729,E2 -16571.729} C_VEL
LIN {X 0,Y 295.762,Z 433.779,A -85,B 0,C 180,E1 -16573.75,E2 -16573.75} C_VEL
LIN {X 0,Y 297.563,Z 428.513,A -85,B 0,C 180,E1 -16575.413,E2 -16575.413} C_VEL
LIN {X 0,Y 299.592,Z 421.877,A -85,B 0,C 180,E1 -16577.055,E2 -16577.055} C_VEL
LIN {X 0,Y 301.329,Z 415.325,A -85,B 0,C 180,E1 -16578.356,E2 -16578.356} C_VEL
LIN {X 0,Y 303.729,Z 405.237,A -85,B 0,C 180,E1 -16579.96,E2 -16579.96} C_VEL
LIN {X 0,Y 305.833,Z 394.972,A -85,B 0,C 180,E1 -16581.223,E2 -16581.223} C_VEL
LIN {X 0,Y 307.511,Z 385.118,A -85,B 0,C 180,E1 -16582.158,E2 -16582.158} C_VEL
LIN {X 0,Y 308.934,Z 374.677,A -85,B 0,C 180,E1 -16582.932,E2 -16582.932} C_VEL
LIN {X 0,Y 310.247,Z 361.9,A -85,B 0,C 180,E1 -16583.58,E2 -16583.58} C_VEL
LIN {X 0,Y 313.884,Z 323.615,A -85,B 0,C 180,E1 -16585.158,E2 -16585.158} C_VEL
LIN {X 0,Y 309.486,Z 314.349,A -85,B 0,C 180,E1 -16586.665,E2 -16586.665} C_VEL
LIN {X 0,Y 305.761,Z 307.795,A -85,B 0,C 180,E1 -16587.998,E2 -16587.998} C_VEL
LIN {X 0,Y 303.002,Z 303.288,A -85,B 0,C 180,E1 -16589.084,E2 -16589.084} C_VEL
LIN {X 0,Y 300.406,Z 299.385,A -85,B 0,C 180,E1 -16590.164,E2 -16590.164} C_VEL
LIN {X 0,Y 297.282,Z 294.926,A -85,B 0,C 180,E1 -16591.589,E2 -16591.589} C_VEL
LIN {X 0,Y 293.95,Z 290.341,A -85,B 0,C 180,E1 -16593.364,E2 -16593.364} C_VEL
LIN {X 0,Y 293.094,Z 287.795,A -85,B 0,C 180,E1 -16595.385,E2 -16595.385} C_VEL
LIN {X 0,Y 291.345,Z 284.007,A -85,B 0,C 180,E1 -16599.677,E2 -16599.677} C_VEL
LIN {X 0,Y 291.3,Z 284.01,A -85,B 0,C 180,E1 -16603.631,E2 -16603.631} C_VEL
LIN {X 0,Y 291.311,Z 284.007,A -85,B 0,C 180,E1 -16607.506,E2 -16607.506} C_VEL
LIN {X 0,Y 291.36,Z 284.118,A -85,B 0,C 180,E1 -16609.523,E2 -16609.523} C_VEL
LIN {X 0,Y 292.595,Z 287.173,A -85,B 0,C 180,E1 -16612.438,E2 -16612.438} C_VEL
LIN {X 0,Y 294.14,Z 289.625,A -85,B 0,C 180,E1 -16614.333,E2 -16614.333} C_VEL
LIN {X 0,Y 294.708,Z 290.99,A -85,B 0,C 180,E1 -16615.086,E2 -16615.086} C_VEL
LIN {X 0,Y 296.054,Z 292.708,A -85,B 0,C 180,E1 -16616.192,E2 -16616.192} C_VEL
LIN {X 0,Y 298.772,Z 297.972,A -85,B 0,C 180,E1 -16618.474,E2 -16618.474} C_VEL
LIN {X 0,Y 304.211,Z 305.838,A -85,B 0,C 180,E1 -16620.722,E2 -16620.722} C_VEL
LIN {X 0,Y 306.221,Z 311.081,A -85,B 0,C 180,E1 -16621.632,E2 -16621.632} C_VEL
LIN {X 0,Y 307.595,Z 315.869,A -85,B 0,C 180,E1 -16622.295,E2 -16622.295} C_VEL
LIN {X 0,Y 309.325,Z 327.507,A -85,B 0,C 180,E1 -16623.468,E2 -16623.468} C_VEL
LIN {X 0,Y 310.843,Z 344.136,A -85,B 0,C 180,E1 -16624.81,E2 -16624.81} C_VEL
LIN {X 0,Y 311.196,Z 354.821,A -85,B 0,C 180,E1 -16625.523,E2 -16625.523} C_VEL
LIN {X 0,Y 307.905,Z 390.527,A -85,B 0,C 180,E1 -16627.038,E2 -16627.038} C_VEL
LIN {X 0,Y 306.112,Z 402.051,A -85,B 0,C 180,E1 -16627.739,E2 -16627.739} C_VEL
LIN {X 0,Y 304.022,Z 413.009,A -85,B 0,C 180,E1 -16628.648,E2 -16628.648} C_VEL
LIN {X 0,Y 301.6,Z 424.272,A -85,B 0,C 180,E1 -16629.897,E2 -16629.897} C_VEL
LIN {X 0,Y 299.684,Z 432.157,A -85,B 0,C 180,E1 -16631.011,E2 -16631.011} C_VEL
LIN {X 0,Y 297.452,Z 440.51,A -85,B 0,C 180,E1 -16632.467,E2 -16632.467} C_VEL
LIN {X 0,Y 295.437,Z 448.031,A -85,B 0,C 180,E1 -16634.123,E2 -16634.123} C_VEL
LIN {X 0,Y 293.647,Z 454.058,A -85,B 0,C 180,E1 -16635.799,E2 -16635.799} C_VEL
LIN {X 0,Y 292.264,Z 458.863,A -85,B 0,C 180,E1 -16637.501,E2 -16637.501} C_VEL
LIN {X 0,Y 290.983,Z 463.265,A -85,B 0,C 180,E1 -16639.563,E2 -16639.563} C_VEL
LIN {X 0,Y 290.109,Z 466.4,A -85,B 0,C 180,E1 -16641.642,E2 -16641.642} C_VEL
LIN {X 0,Y 289.734,Z 467.728,A -85,B 0,C 180,E1 -16643.034,E2 -16643.034} C_VEL
LIN {X 0,Y 289.568,Z 468.552,A -85,B 0,C 180,E1 -16644.429,E2 -16644.429} C_VEL
LIN {X 0,Y 289.536,Z 468.88,A -85,B 0,C 180,E1 -16645.824,E2 -16645.824} C_VEL
LIN {X 0,Y 289.544,Z 468.807,A -85,B 0,C 180,E1 -16647.391,E2 -16647.391} C_VEL
LIN {X 0,Y 289.557,Z 470.046,A -85,B 0,C 180,E1 -16648.609,E2 -16648.609} C_VEL
LIN {X 0,Y 289.586,Z 470.976,A -85,B 0,C 180,E1 -16650,E2 -16650} C_VEL
LIN {X 0,Y 289.506,Z 471.302,A -85,B 0,C 180,E1 -16651.391,E2 -16651.391} C_VEL
LIN {X 0,Y 289.519,Z 471.152,A -85,B 0,C 180,E1 -16652.783,E2 -16652.783} C_VEL
LIN {X 0,Y 289.505,Z 470.541,A -85,B 0,C 180,E1 -16654.176,E2 -16654.176} C_VEL
LIN {X 0,Y 289.528,Z 469.463,A -85,B 0,C 180,E1 -16655.572,E2 -16655.572} C_VEL
LIN {X 0,Y 289.864,Z 466.747,A -85,B 0,C 180,E1 -16657.663,E2 -16657.663} C_VEL
LIN {X 0,Y 290.275,Z 464.327,A -85,B 0,C 180,E1 -16659.054,E2 -16659.054} C_VEL
LIN {X 0,Y 291.153,Z 459.406,A -85,B 0,C 180,E1 -16661.134,E2 -16661.134} C_VEL
LIN {X 0,Y 292.209,Z 454.147,A -85,B 0,C 180,E1 -16662.854,E2 -16662.854} C_VEL
LIN {X 0,Y 293.195,Z 449.013,A -85,B 0,C 180,E1 -16664.223,E2 -16664.223} C_VEL
LIN {X 0,Y 294.371,Z 442.854,A -85,B 0,C 180,E1 -16665.58,E2 -16665.58} C_VEL
LIN {X 0,Y 295.68,Z 436.395,A -85,B 0,C 180,E1 -16666.75,E2 -16666.75} C_VEL
LIN {X 0,Y 296.904,Z 428.611,A -85,B 0,C 180,E1 -16667.922,E2 -16667.922} C_VEL
LIN {X 0,Y 298.293,Z 420.403,A -85,B 0,C 180,E1 -16668.902,E2 -16668.902} C_VEL
LIN {X 0,Y 299.387,Z 411.881,A -85,B 0,C 180,E1 -16669.721,E2 -16669.721} C_VEL
LIN {X 0,Y 300.764,Z 400.616,A -85,B 0,C 180,E1 -16670.518,E2 -16670.518} C_VEL
LIN {X 0,Y 301.572,Z 389.412,A -85,B 0,C 180,E1 -16671.03,E2 -16671.03} C_VEL
LIN {X 0,Y 302.326,Z 364.302,A -85,B 0,C 180,E1 -16671.682,E2 -16671.682} C_VEL
LIN {X 0,Y 302.525,Z 350.941,A -85,B 0,C 180,E1 -16672.017,E2 -16672.017} C_VEL
LIN {X 0,Y 299.907,Z 333.477,A -85,B 0,C 180,E1 -16672.738,E2 -16672.738} C_VEL
LIN {X 0,Y 295.986,Z 314.305,A -85,B 0,C 180,E1 -16673.658,E2 -16673.658} C_VEL
LIN {X 0,Y 295.012,Z 309.488,A -85,B 0,C 180,E1 -16673.937,E2 -16673.937} C_VEL
LIN {X 0,Y 295.597,Z 304.937,A -85,B 0,C 180,E1 -16675.376,E2 -16675.376} C_VEL
LIN {X 0,Y 294.443,Z 297.534,A -85,B 0,C 180,E1 -16677.971,E2 -16677.971} C_VEL
LIN {X 0,Y 292.558,Z 289.13,A -85,B 0,C 180,E1 -16681.096,E2 -16681.096} C_VEL
LIN {X 0,Y 291.344,Z 284.002,A -85,B 0,C 180,E1 -16683.168,E2 -16683.168} C_VEL
LIN {X 0,Y 291.399,Z 283.996,A -85,B 0,C 180,E1 -16687.081,E2 -16687.081} C_VEL
LIN {X 0,Y 291.34,Z 284.007,A -85,B 0,C 180,E1 -16690.641,E2 -16690.641} C_VEL
LIN {X 0,Y 291.3,Z 284.006,A -85,B 0,C 180,E1 -16694.4,E2 -16694.4} C_VEL
LIN {X 0,Y 291.304,Z 284.01,A -85,B 0,C 180,E1 -16698.409,E2 -16698.409} C_VEL
LIN {X 0,Y 291.404,Z 283.998,A -85,B 0,C 180,E1 -16702.915,E2 -16702.915} C_VEL
LIN {X 0,Y 291.352,Z 284.004,A -85,B 0,C 180,E1 -16706.299,E2 -16706.299} C_VEL
LIN {X 0,Y 291.376,Z 284.001,A -85,B 0,C 180,E1 -16710.264,E2 -16710.264} C_VEL
LIN {X 0,Y 291.381,Z 283.995,A -85,B 0,C 180,E1 -16714.265,E2 -16714.265} C_VEL
LIN {X 0,Y 291.377,Z 284,A -85,B 0,C 180,E1 -16717.295,E2 -16717.295} C_VEL
LIN {X 0,Y 291.445,Z 283.993,A -85,B 0,C 180,E1 -16720.265,E2 -16720.265} C_VEL
LIN {X 0,Y 291.502,Z 283.978,A -85,B 0,C 180,E1 -16724.661,E2 -16724.661} C_VEL
LIN {X 0,Y 291.539,Z 283.965,A -85,B 0,C 180,E1 -16728.877,E2 -16728.877} C_VEL
LIN {X 0,Y 291.691,Z 283.959,A -85,B 0,C 180,E1 -16731.684,E2 -16731.684} C_VEL
LIN {X 0,Y 291.624,Z 283.955,A -85,B 0,C 180,E1 -16734.464,E2 -16734.464} C_VEL
LIN {X 0,Y 291.885,Z 283.928,A -85,B 0,C 180,E1 -16738.616,E2 -16738.616} C_VEL
LIN {X 0,Y 291.885,Z 283.93,A -85,B 0,C 180,E1 -16741.375,E2 -16741.375} C_VEL
LIN {X 0,Y 291.656,Z 283.959,A -85,B 0,C 180,E1 -16746.562,E2 -16746.562} C_VEL
LIN {X 0,Y 291.564,Z 283.972,A -85,B 0,C 180,E1 -16749.709,E2 -16749.709} C_VEL
LIN {X 0,Y 291.516,Z 283.986,A -85,B 0,C 180,E1 -16753.945,E2 -16753.945} C_VEL
LIN {X 0,Y 291.48,Z 283.986,A -85,B 0,C 180,E1 -16756.813,E2 -16756.813} C_VEL
LIN {X 0,Y 291.442,Z 283.988,A -85,B 0,C 180,E1 -16759.87,E2 -16759.87} C_VEL
LIN {X 0,Y 291.389,Z 283.995,A -85,B 0,C 180,E1 -16764.2,E2 -16764.2} C_VEL
LIN {X 0,Y 291.408,Z 283.996,A -85,B 0,C 180,E1 -16767.267,E2 -16767.267} C_VEL
LIN {X 0,Y 291.319,Z 284.011,A -85,B 0,C 180,E1 -16770.433,E2 -16770.433} C_VEL
LIN {X 0,Y 291.328,Z 284.008,A -85,B 0,C 180,E1 -16773.694,E2 -16773.694} C_VEL
LIN {X 0,Y 291.37,Z 283.997,A -85,B 0,C 180,E1 -16777.253,E2 -16777.253} C_VEL
LIN {X 0,Y 291.382,Z 283.992,A -85,B 0,C 180,E1 -16780.627,E2 -16780.627} C_VEL
LIN {X 0,Y 291.385,Z 283.995,A -85,B 0,C 180,E1 -16784.375,E2 -16784.375} C_VEL
LIN {X 0,Y 291.416,Z 284.052,A -85,B 0,C 180,E1 -16787.905,E2 -16787.905} C_VEL
LIN {X 0,Y 291.916,Z 286.399,A -85,B 0,C 180,E1 -16788.795,E2 -16788.795} C_VEL
LIN {X 0,Y 299.766,Z 303.491,A -85,B 0,C 180,E1 -16790.115,E2 -16790.115} C_VEL
LIN {X 0,Y 303.505,Z 313.146,A -85,B 0,C 180,E1 -16790.749,E2 -16790.749} C_VEL
LIN {X 0,Y 302.242,Z 362.724,A -85,B 0,C 180,E1 -16791.989,E2 -16791.989} C_VEL
LIN {X 0,Y 301.724,Z 372.664,A -85,B 0,C 180,E1 -16792.42,E2 -16792.42} C_VEL
LIN {X 0,Y 300.785,Z 384.683,A -85,B 0,C 180,E1 -16793.22,E2 -16793.22} C_VEL
LIN {X 0,Y 299.636,Z 394.089,A -85,B 0,C 180,E1 -16794.1,E2 -16794.1} C_VEL
LIN {X 0,Y 298.457,Z 402.969,A -85,B 0,C 180,E1 -16795.178,E2 -16795.178} C_VEL
LIN {X 0,Y 297.32,Z 410.171,A -85,B 0,C 180,E1 -16796.256,E2 -16796.256} C_VEL
LIN {X 0,Y 296.193,Z 416.189,A -85,B 0,C 180,E1 -16797.33,E2 -16797.33} C_VEL
LIN {X 0,Y 295.207,Z 421.347,A -85,B 0,C 180,E1 -16798.416,E2 -16798.416} C_VEL
LIN {X 0,Y 294.026,Z 427.062,A -85,B 0,C 180,E1 -16799.871,E2 -16799.871} C_VEL
LIN {X 0,Y 293.021,Z 431.772,A -85,B 0,C 180,E1 -16801.335,E2 -16801.335} C_VEL
LIN {X 0,Y 292.073,Z 435.841,A -85,B 0,C 180,E1 -16802.899,E2 -16802.899} C_VEL
LIN {X 0,Y 291.411,Z 438.738,A -85,B 0,C 180,E1 -16804.272,E2 -16804.272} C_VEL
LIN {X 0,Y 290.784,Z 441.134,A -85,B 0,C 180,E1 -16805.74,E2 -16805.74} C_VEL
LIN {X 0,Y 290.324,Z 442.868,A -85,B 0,C 180,E1 -16807.212,E2 -16807.212} C_VEL
LIN {X 0,Y 289.911,Z 444.032,A -85,B 0,C 180,E1 -16808.677,E2 -16808.677} C_VEL
LIN {X 0,Y 289.518,Z 444.851,A -85,B 0,C 180,E1 -16811.192,E2 -16811.192} C_VEL
LIN {X 0,Y 289.385,Z 444.361,A -85,B 0,C 180,E1 -16813.057,E2 -16813.057} C_VEL
LIN {X 0,Y 289.435,Z 443.342,A -85,B 0,C 180,E1 -16814.509,E2 -16814.509} C_VEL
LIN {X 0,Y 289.536,Z 441.551,A -85,B 0,C 180,E1 -16816.124,E2 -16816.124} C_VEL
LIN {X 0,Y 289.879,Z 438.403,A -85,B 0,C 180,E1 -16818.108,E2 -16818.108} C_VEL
LIN {X 0,Y 290.286,Z 433.523,A -85,B 0,C 180,E1 -16820.243,E2 -16820.243} C_VEL
LIN {X 0,Y 290.718,Z 429.42,A -85,B 0,C 180,E1 -16821.66,E2 -16821.66} C_VEL
LIN {X 0,Y 291.247,Z 423.047,A -85,B 0,C 180,E1 -16823.419,E2 -16823.419} C_VEL
LIN {X 0,Y 291.881,Z 416.777,A -85,B 0,C 180,E1 -16824.82,E2 -16824.82} C_VEL
LIN {X 0,Y 292.512,Z 410.186,A -85,B 0,C 180,E1 -16826.039,E2 -16826.039} C_VEL
LIN {X 0,Y 293.246,Z 402.196,A -85,B 0,C 180,E1 -16827.253,E2 -16827.253} C_VEL
LIN {X 0,Y 294.104,Z 392.203,A -85,B 0,C 180,E1 -16828.46,E2 -16828.46} C_VEL
LIN {X 0,Y 294.777,Z 381.539,A -85,B 0,C 180,E1 -16829.412,E2 -16829.412} C_VEL
LIN {X 0,Y 295.238,Z 371.756,A -85,B 0,C 180,E1 -16830.042,E2 -16830.042} C_VEL
LIN {X 0,Y 295.476,Z 362.466,A -85,B 0,C 180,E1 -16830.457,E2 -16830.457} C_VEL
LIN {X 0,Y 296.404,Z 307.996,A -85,B 0,C 180,E1 -16831.816,E2 -16831.816} C_VEL
LIN {X 0,Y 293.344,Z 289.953,A -85,B 0,C 180,E1 -16832.425,E2 -16832.425} C_VEL
LIN {X 0,Y 291.989,Z 285.307,A -85,B 0,C 180,E1 -16832.63,E2 -16832.63} C_VEL
LIN {X 0,Y 291.648,Z 283.972,A -85,B 0,C 180,E1 -16833.195,E2 -16833.195} C_VEL
LIN {X 0,Y 291.702,Z 283.963,A -85,B 0,C 180,E1 -16836.919,E2 -16836.919} C_VEL
LIN {X 0,Y 291.542,Z 283.981,A -85,B 0,C 180,E1 -16839.715,E2 -16839.715} C_VEL
LIN {X 0,Y 291.485,Z 283.987,A -85,B 0,C 180,E1 -16843.952,E2 -16843.952} C_VEL
LIN {X 0,Y 291.441,Z 283.991,A -85,B 0,C 180,E1 -16848.27,E2 -16848.27} C_VEL
LIN {X 0,Y 291.345,Z 284.007,A -85,B 0,C 180,E1 -16851.214,E2 -16851.214} C_VEL
LIN {X 0,Y 291.334,Z 284.005,A -85,B 0,C 180,E1 -16854.211,E2 -16854.211} C_VEL
LIN {X 0,Y 291.325,Z 284.01,A -85,B 0,C 180,E1 -16857.282,E2 -16857.282} C_VEL
LIN {X 0,Y 291.291,Z 284.008,A -85,B 0,C 180,E1 -16860.443,E2 -16860.443} C_VEL
LIN {X 0,Y 291.317,Z 284.01,A -85,B 0,C 180,E1 -16863.702,E2 -16863.702} C_VEL
LIN {X 0,Y 291.328,Z 284.007,A -85,B 0,C 180,E1 -16867.252,E2 -16867.252} C_VEL
LIN {X 0,Y 291.277,Z 284.011,A -85,B 0,C 180,E1 -16870.652,E2 -16870.652} C_VEL
LIN {X 0,Y 291.261,Z 284.013,A -85,B 0,C 180,E1 -16874.408,E2 -16874.408} C_VEL
LIN {X 0,Y 291.307,Z 284.008,A -85,B 0,C 180,E1 -16878.409,E2 -16878.409} C_VEL
LIN {X 0,Y 291.346,Z 284.003,A -85,B 0,C 180,E1 -16881.165,E2 -16881.165} C_VEL
LIN {X 0,Y 291.346,Z 284.003,A -85,B 0,C 180,E1 -16884.631,E2 -16884.631} C_VEL
LIN {X 0,Y 291.352,Z 284.007,A -85,B 0,C 180,E1 -16887.955,E2 -16887.955} C_VEL
LIN {X 0,Y 291.332,Z 284.005,A -85,B 0,C 180,E1 -16891.159,E2 -16891.159} C_VEL
LIN {X 0,Y 291.351,Z 284.004,A -85,B 0,C 180,E1 -16894.272,E2 -16894.272} C_VEL
LIN {X 0,Y 291.362,Z 283.998,A -85,B 0,C 180,E1 -16897.304,E2 -16897.304} C_VEL
LIN {X 0,Y 291.467,Z 283.976,A -85,B 0,C 180,E1 -16900.904,E2 -16900.904} C_VEL
LIN {X 0,Y 291.346,Z 284.573,A -85,B 0,C 180,E1 -16901.414,E2 -16901.414} C_VEL
LIN {X 0,Y 290.88,Z 286.644,A -85,B 0,C 180,E1 -16901.995,E2 -16901.995} C_VEL
LIN {X 0,Y 290.027,Z 290.449,A -85,B 0,C 180,E1 -16902.549,E2 -16902.549} C_VEL
LIN {X 0,Y 288.811,Z 296.105,A -85,B 0,C 180,E1 -16902.972,E2 -16902.972} C_VEL
LIN {X 0,Y 287.183,Z 304.9,A -85,B 0,C 180,E1 -16903.315,E2 -16903.315} C_VEL
LIN {X 0,Y 286.878,Z 311.612,A -85,B 0,C 180,E1 -16903.568,E2 -16903.568} C_VEL
LIN {X 0,Y 285.604,Z 364.117,A -85,B 0,C 180,E1 -16905.623,E2 -16905.623} C_VEL
LIN {X 0,Y 285.27,Z 375.18,A -85,B 0,C 180,E1 -16906.288,E2 -16906.288} C_VEL
LIN {X 0,Y 284.855,Z 386.029,A -85,B 0,C 180,E1 -16907.176,E2 -16907.176} C_VEL
LIN {X 0,Y 284.433,Z 395.824,A -85,B 0,C 180,E1 -16908.243,E2 -16908.243} C_VEL
LIN {X 0,Y 283.931,Z 404.943,A -85,B 0,C 180,E1 -16909.487,E2 -16909.487} C_VEL
LIN {X 0,Y 283.425,Z 414.434,A -85,B 0,C 180,E1 -16911.089,E2 -16911.089} C_VEL
LIN {X 0,Y 283.049,Z 422.649,A -85,B 0,C 180,E1 -16912.873,E2 -16912.873} C_VEL
LIN {X 0,Y 282.757,Z 428.043,A -85,B 0,C 180,E1 -16914.299,E2 -16914.299} C_VEL
LIN {X 0,Y 282.754,Z 432.571,A -85,B 0,C 180,E1 -16915.728,E2 -16915.728} C_VEL
LIN {X 0,Y 282.55,Z 436.302,A -85,B 0,C 180,E1 -16917.153,E2 -16917.153} C_VEL
LIN {X 0,Y 282.413,Z 440.625,A -85,B 0,C 180,E1 -16919.292,E2 -16919.292} C_VEL
LIN {X 0,Y 282.538,Z 443.632,A -85,B 0,C 180,E1 -16921.43,E2 -16921.43} C_VEL
LIN {X 0,Y 282.77,Z 444.84,A -85,B 0,C 180,E1 -16922.854,E2 -16922.854} C_VEL
LIN {X 0,Y 283.164,Z 445.53,A -85,B 0,C 180,E1 -16924.275,E2 -16924.275} C_VEL
LIN {X 0,Y 283.623,Z 445.719,A -85,B 0,C 180,E1 -16925.693,E2 -16925.693} C_VEL
LIN {X 0,Y 284.049,Z 445.419,A -85,B 0,C 180,E1 -16927.111,E2 -16927.111} C_VEL
LIN {X 0,Y 284.576,Z 444.577,A -85,B 0,C 180,E1 -16928.526,E2 -16928.526} C_VEL
LIN {X 0,Y 286.172,Z 441.927,A -85,B 0,C 180,E1 -16930.78,E2 -16930.78} C_VEL
LIN {X 0,Y 287.723,Z 438.517,A -85,B 0,C 180,E1 -16932.704,E2 -16932.704} C_VEL
LIN {X 0,Y 289.035,Z 435.313,A -85,B 0,C 180,E1 -16934.077,E2 -16934.077} C_VEL
LIN {X 0,Y 290.926,Z 430.272,A -85,B 0,C 180,E1 -16935.774,E2 -16935.774} C_VEL
LIN {X 0,Y 293.04,Z 424.007,A -85,B 0,C 180,E1 -16937.449,E2 -16937.449} C_VEL
LIN {X 0,Y 295.387,Z 416.22,A -85,B 0,C 180,E1 -16939.1,E2 -16939.1} C_VEL
LIN {X 0,Y 297.672,Z 407.379,A -85,B 0,C 180,E1 -16940.564,E2 -16940.564} C_VEL
LIN {X 0,Y 299.902,Z 397.653,A -85,B 0,C 180,E1 -16941.844,E2 -16941.844} C_VEL
LIN {X 0,Y 301.981,Z 386.584,A -85,B 0,C 180,E1 -16942.947,E2 -16942.947} C_VEL
LIN {X 0,Y 303.491,Z 376.607,A -85,B 0,C 180,E1 -16943.729,E2 -16943.729} C_VEL
LIN {X 0,Y 305.079,Z 363.291,A -85,B 0,C 180,E1 -16944.456,E2 -16944.456} C_VEL
LIN {X 0,Y 308.768,Z 326.477,A -85,B 0,C 180,E1 -16946.009,E2 -16946.009} C_VEL
LIN {X 0,Y 304.513,Z 317.338,A -85,B 0,C 180,E1 -16947.617,E2 -16947.617} C_VEL
LIN {X 0,Y 300.09,Z 309.658,A -85,B 0,C 180,E1 -16949.391,E2 -16949.391} C_VEL
LIN {X 0,Y 297.263,Z 305.268,A -85,B 0,C 180,E1 -16950.643,E2 -16950.643} C_VEL
LIN {X 0,Y 294.473,Z 301.108,A -85,B 0,C 180,E1 -16952.008,E2 -16952.008} C_VEL
LIN {X 0,Y 291.155,Z 296.45,A -85,B 0,C 180,E1 -16953.883,E2 -16953.883} C_VEL
LIN {X 0,Y 287.804,Z 292.349,A -85,B 0,C 180,E1 -16956.156,E2 -16956.156} C_VEL
LIN {X 0,Y 287.069,Z 291.395,A -85,B 0,C 180,E1 -16956.859,E2 -16956.859} C_VEL
LIN {X 0,Y 286.355,Z 289.082,A -85,B 0,C 180,E1 -16959.656,E2 -16959.656} C_VEL
LIN {X 0,Y 285.502,Z 288.093,A -85,B 0,C 180,E1 -16963.575,E2 -16963.575} C_VEL
LIN {X 0,Y 285.735,Z 288.368,A -85,B 0,C 180,E1 -16966.473,E2 -16966.473} C_VEL
LIN {X 0,Y 286.85,Z 289.582,A -85,B 0,C 180,E1 -16969.426,E2 -16969.426} C_VEL
LIN {X 0,Y 289.022,Z 293.891,A -85,B 0,C 180,E1 -16973.369,E2 -16973.369} C_VEL
LIN {X 0,Y 290.753,Z 297.043,A -85,B 0,C 180,E1 -16975.274,E2 -16975.274} C_VEL
LIN {X 0,Y 292.538,Z 299.432,A -85,B 0,C 180,E1 -16976.334,E2 -16976.334} C_VEL
LIN {X 0,Y 296.603,Z 305.27,A -85,B 0,C 180,E1 -16978.421,E2 -16978.421} C_VEL
LIN {X 0,Y 300.772,Z 311.573,A -85,B 0,C 180,E1 -16980.238,E2 -16980.238} C_VEL
LIN {X 0,Y 302.472,Z 316.605,A -85,B 0,C 180,E1 -16981.08,E2 -16981.08} C_VEL
LIN {X 0,Y 303.361,Z 320.311,A -85,B 0,C 180,E1 -16981.591,E2 -16981.591} C_VEL
LIN {X 0,Y 304.917,Z 332.528,A -85,B 0,C 180,E1 -16982.831,E2 -16982.831} C_VEL
LIN {X 0,Y 306.083,Z 350.933,A -85,B 0,C 180,E1 -16984.309,E2 -16984.309} C_VEL
LIN {X 0,Y 305.961,Z 357.993,A -85,B 0,C 180,E1 -16984.721,E2 -16984.721} C_VEL
LIN {X 0,Y 302.652,Z 389.919,A -85,B 0,C 180,E1 -16986.113,E2 -16986.113} C_VEL
LIN {X 0,Y 300.684,Z 401.918,A -85,B 0,C 180,E1 -16986.861,E2 -16986.861} C_VEL
LIN {X 0,Y 298.649,Z 412.01,A -85,B 0,C 180,E1 -16987.699,E2 -16987.699} C_VEL
LIN {X 0,Y 296.065,Z 423.35,A -85,B 0,C 180,E1 -16988.959,E2 -16988.959} C_VEL
LIN {X 0,Y 293.918,Z 431.258,A -85,B 0,C 180,E1 -16990.078,E2 -16990.078} C_VEL
LIN {X 0,Y 291.323,Z 440.493,A -85,B 0,C 180,E1 -16991.722,E2 -16991.722} C_VEL
LIN {X 0,Y 289.088,Z 447.941,A -85,B 0,C 180,E1 -16993.402,E2 -16993.402} C_VEL
LIN {X 0,Y 287.223,Z 453.833,A -85,B 0,C 180,E1 -16995.112,E2 -16995.112} C_VEL
LIN {X 0,Y 285.354,Z 459.405,A -85,B 0,C 180,E1 -16997.193,E2 -16997.193} C_VEL
LIN {X 0,Y 284.428,Z 462.321,A -85,B 0,C 180,E1 -16998.599,E2 -16998.599} C_VEL
LIN {X 0,Y 283.662,Z 464.663,A -85,B 0,C 180,E1 -17000.012,E2 -17000.012} C_VEL
LIN {X 0,Y 283.078,Z 466.457,A -85,B 0,C 180,E1 -17001.433,E2 -17001.433} C_VEL
LIN {X 0,Y 282.685,Z 467.646,A -85,B 0,C 180,E1 -17002.859,E2 -17002.859} C_VEL
LIN {X 0,Y 282.492,Z 468.318,A -85,B 0,C 180,E1 -17004.376,E2 -17004.376} C_VEL
LIN {X 0,Y 282.463,Z 468.169,A -85,B 0,C 180,E1 -17006.969,E2 -17006.969} C_VEL
LIN {X 0,Y 282.474,Z 469.641,A -85,B 0,C 180,E1 -17008.574,E2 -17008.574} C_VEL
LIN {X 0,Y 282.499,Z 470.585,A -85,B 0,C 180,E1 -17010,E2 -17010} C_VEL
LIN {X 0,Y 282.426,Z 470.948,A -85,B 0,C 180,E1 -17011.426,E2 -17011.426} C_VEL
LIN {X 0,Y 282.445,Z 470.85,A -85,B 0,C 180,E1 -17012.852,E2 -17012.852} C_VEL
LIN {X 0,Y 282.408,Z 470.291,A -85,B 0,C 180,E1 -17014.281,E2 -17014.281} C_VEL
LIN {X 0,Y 282.454,Z 469.251,A -85,B 0,C 180,E1 -17015.712,E2 -17015.712} C_VEL
LIN {X 0,Y 282.802,Z 466.611,A -85,B 0,C 180,E1 -17017.856,E2 -17017.856} C_VEL
LIN {X 0,Y 283.235,Z 464.238,A -85,B 0,C 180,E1 -17019.281,E2 -17019.281} C_VEL
LIN {X 0,Y 284.168,Z 459.406,A -85,B 0,C 180,E1 -17021.411,E2 -17021.411} C_VEL
LIN {X 0,Y 285.269,Z 454.222,A -85,B 0,C 180,E1 -17023.172,E2 -17023.172} C_VEL
LIN {X 0,Y 286.326,Z 449.171,A -85,B 0,C 180,E1 -17024.571,E2 -17024.571} C_VEL
LIN {X 0,Y 287.564,Z 443.109,A -85,B 0,C 180,E1 -17025.959,E2 -17025.959} C_VEL
LIN {X 0,Y 289.092,Z 435.749,A -85,B 0,C 180,E1 -17027.326,E2 -17027.326} C_VEL
LIN {X 0,Y 290.435,Z 427.897,A -85,B 0,C 180,E1 -17028.518,E2 -17028.518} C_VEL
LIN {X 0,Y 291.838,Z 419.61,A -85,B 0,C 180,E1 -17029.52,E2 -17029.52} C_VEL
LIN {X 0,Y 293.268,Z 409.086,A -85,B 0,C 180,E1 -17030.516,E2 -17030.516} C_VEL
LIN {X 0,Y 294.539,Z 397.881,A -85,B 0,C 180,E1 -17031.239,E2 -17031.239} C_VEL
LIN {X 0,Y 295.258,Z 388.162,A -85,B 0,C 180,E1 -17031.661,E2 -17031.661} C_VEL
LIN {X 0,Y 296.194,Z 351.761,A -85,B 0,C 180,E1 -17032.61,E2 -17032.61} C_VEL
LIN {X 0,Y 293.701,Z 335.152,A -85,B 0,C 180,E1 -17033.321,E2 -17033.321} C_VEL
LIN {X 0,Y 290.163,Z 317.476,A -85,B 0,C 180,E1 -17034.196,E2 -17034.196} C_VEL
LIN {X 0,Y 288.354,Z 309.228,A -85,B 0,C 180,E1 -17034.645,E2 -17034.645} C_VEL
LIN {X 0,Y 288.622,Z 305.154,A -85,B 0,C 180,E1 -17035.995,E2 -17035.995} C_VEL
LIN {X 0,Y 287.267,Z 297.731,A -85,B 0,C 180,E1 -17038.702,E2 -17038.702} C_VEL
LIN {X 0,Y 285.305,Z 289.269,A -85,B 0,C 180,E1 -17041.979,E2 -17041.979} C_VEL
LIN {X 0,Y 284.319,Z 284.885,A -85,B 0,C 180,E1 -17043.79,E2 -17043.79} C_VEL
LIN {X 0,Y 284.318,Z 284.885,A -85,B 0,C 180,E1 -17047.716,E2 -17047.716} C_VEL
LIN {X 0,Y 284.316,Z 284.883,A -85,B 0,C 180,E1 -17049.993,E2 -17049.993} C_VEL
LIN {X 0,Y 284.255,Z 284.884,A -85,B 0,C 180,E1 -17054.188,E2 -17054.188} C_VEL
LIN {X 0,Y 284.249,Z 284.887,A -85,B 0,C 180,E1 -17058.116,E2 -17058.116} C_VEL
LIN {X 0,Y 284.313,Z 284.881,A -85,B 0,C 180,E1 -17062.28,E2 -17062.28} C_VEL
LIN {X 0,Y 284.315,Z 284.874,A -85,B 0,C 180,E1 -17065.348,E2 -17065.348} C_VEL
LIN {X 0,Y 284.293,Z 284.876,A -85,B 0,C 180,E1 -17068.721,E2 -17068.721} C_VEL
LIN {X 0,Y 284.296,Z 284.882,A -85,B 0,C 180,E1 -17071.982,E2 -17071.982} C_VEL
LIN {X 0,Y 284.332,Z 284.88,A -85,B 0,C 180,E1 -17076.142,E2 -17076.142} C_VEL
LIN {X 0,Y 284.382,Z 284.868,A -85,B 0,C 180,E1 -17079.901,E2 -17079.901} C_VEL
LIN {X 0,Y 284.452,Z 284.855,A -85,B 0,C 180,E1 -17084.488,E2 -17084.488} C_VEL
LIN {X 0,Y 284.491,Z 284.844,A -85,B 0,C 180,E1 -17088.597,E2 -17088.597} C_VEL
LIN {X 0,Y 284.642,Z 284.835,A -85,B 0,C 180,E1 -17091.476,E2 -17091.476} C_VEL
LIN {X 0,Y 284.595,Z 284.83,A -85,B 0,C 180,E1 -17094.327,E2 -17094.327} C_VEL
LIN {X 0,Y 284.851,Z 284.804,A -85,B 0,C 180,E1 -17098.582,E2 -17098.582} C_VEL
LIN {X 0,Y 284.851,Z 284.806,A -85,B 0,C 180,E1 -17101.409,E2 -17101.409} C_VEL
LIN {X 0,Y 284.65,Z 284.836,A -85,B 0,C 180,E1 -17107.086,E2 -17107.086} C_VEL
LIN {X 0,Y 284.51,Z 284.849,A -85,B 0,C 180,E1 -17109.952,E2 -17109.952} C_VEL
LIN {X 0,Y 284.476,Z 284.858,A -85,B 0,C 180,E1 -17114.298,E2 -17114.298} C_VEL
LIN {X 0,Y 284.418,Z 284.867,A -85,B 0,C 180,E1 -17117.243,E2 -17117.243} C_VEL
LIN {X 0,Y 284.37,Z 284.867,A -85,B 0,C 180,E1 -17120.237,E2 -17120.237} C_VEL
LIN {X 0,Y 284.358,Z 284.873,A -85,B 0,C 180,E1 -17123.87,E2 -17123.87} C_VEL
LIN {X 0,Y 284.383,Z 284.872,A -85,B 0,C 180,E1 -17127.168,E2 -17127.168} C_VEL
LIN {X 0,Y 284.278,Z 284.882,A -85,B 0,C 180,E1 -17131.27,E2 -17131.27} C_VEL
LIN {X 0,Y 284.324,Z 284.865,A -85,B 0,C 180,E1 -17135.344,E2 -17135.344} C_VEL
LIN {X 0,Y 284.309,Z 284.884,A -85,B 0,C 180,E1 -17138.162,E2 -17138.162} C_VEL
LIN {X 0,Y 284.332,Z 284.882,A -85,B 0,C 180,E1 -17142.139,E2 -17142.139} C_VEL
LIN {X 0,Y 284.331,Z 284.879,A -85,B 0,C 180,E1 -17146.204,E2 -17146.204} C_VEL
LIN {X 0,Y 284.373,Z 285.063,A -85,B 0,C 180,E1 -17147.314,E2 -17147.314} C_VEL
LIN {X 0,Y 284.725,Z 286.597,A -85,B 0,C 180,E1 -17147.963,E2 -17147.963} C_VEL
LIN {X 0,Y 293.533,Z 305.498,A -85,B 0,C 180,E1 -17149.511,E2 -17149.511} C_VEL
LIN {X 0,Y 297.26,Z 314.819,A -85,B 0,C 180,E1 -17150.165,E2 -17150.165} C_VEL
LIN {X 0,Y 295.899,Z 362.841,A -85,B 0,C 180,E1 -17151.383,E2 -17151.383} C_VEL
LIN {X 0,Y 295.393,Z 372.182,A -85,B 0,C 180,E1 -17151.787,E2 -17151.787} C_VEL
LIN {X 0,Y 294.64,Z 382.196,A -85,B 0,C 180,E1 -17152.43,E2 -17152.43} C_VEL
LIN {X 0,Y 293.329,Z 393.322,A -85,B 0,C 180,E1 -17153.417,E2 -17153.417} C_VEL
LIN {X 0,Y 292.076,Z 402.398,A -85,B 0,C 180,E1 -17154.514,E2 -17154.514} C_VEL
LIN {X 0,Y 290.925,Z 409.458,A -85,B 0,C 180,E1 -17155.563,E2 -17155.563} C_VEL
LIN {X 0,Y 289.505,Z 416.798,A -85,B 0,C 180,E1 -17156.893,E2 -17156.893} C_VEL
LIN {X 0,Y 288.223,Z 422.935,A -85,B 0,C 180,E1 -17158.254,E2 -17158.254} C_VEL
LIN {X 0,Y 286.927,Z 428.817,A -85,B 0,C 180,E1 -17159.859,E2 -17159.859} C_VEL
LIN {X 0,Y 285.912,Z 433.261,A -85,B 0,C 180,E1 -17161.359,E2 -17161.359} C_VEL
LIN {X 0,Y 284.912,Z 437.286,A -85,B 0,C 180,E1 -17163.054,E2 -17163.054} C_VEL
LIN {X 0,Y 283.963,Z 440.963,A -85,B 0,C 180,E1 -17165.119,E2 -17165.119} C_VEL
LIN {X 0,Y 283.401,Z 442.846,A -85,B 0,C 180,E1 -17166.623,E2 -17166.623} C_VEL
LIN {X 0,Y 282.959,Z 444.156,A -85,B 0,C 180,E1 -17168.127,E2 -17168.127} C_VEL
LIN {X 0,Y 282.633,Z 444.928,A -85,B 0,C 180,E1 -17169.628,E2 -17169.628} C_VEL
LIN {X 0,Y 282.431,Z 445.174,A -85,B 0,C 180,E1 -17171.126,E2 -17171.126} C_VEL
LIN {X 0,Y 282.319,Z 444.817,A -85,B 0,C 180,E1 -17172.619,E2 -17172.619} C_VEL
LIN {X 0,Y 282.335,Z 443.889,A -85,B 0,C 180,E1 -17174.109,E2 -17174.109} C_VEL
LIN {X 0,Y 282.445,Z 441.969,A -85,B 0,C 180,E1 -17176.003,E2 -17176.003} C_VEL
LIN {X 0,Y 282.832,Z 437.885,A -85,B 0,C 180,E1 -17178.534,E2 -17178.534} C_VEL
LIN {X 0,Y 283.128,Z 434.683,A -85,B 0,C 180,E1 -17179.994,E2 -17179.994} C_VEL
LIN {X 0,Y 283.668,Z 429.655,A -85,B 0,C 180,E1 -17181.784,E2 -17181.784} C_VEL
LIN {X 0,Y 284.091,Z 424.602,A -85,B 0,C 180,E1 -17183.252,E2 -17183.252} C_VEL
LIN {X 0,Y 284.72,Z 418.574,A -85,B 0,C 180,E1 -17184.689,E2 -17184.689} C_VEL
LIN {X 0,Y 285.413,Z 411.242,A -85,B 0,C 180,E1 -17186.117,E2 -17186.117} C_VEL
LIN {X 0,Y 286.169,Z 403.394,A -85,B 0,C 180,E1 -17187.361,E2 -17187.361} C_VEL
LIN {X 0,Y 286.905,Z 395.115,A -85,B 0,C 180,E1 -17188.421,E2 -17188.421} C_VEL
LIN {X 0,Y 287.572,Z 386.476,A -85,B 0,C 180,E1 -17189.3,E2 -17189.3} C_VEL
LIN {X 0,Y 288.115,Z 375.888,A -85,B 0,C 180,E1 -17190.125,E2 -17190.125} C_VEL
LIN {X 0,Y 288.564,Z 363.77,A -85,B 0,C 180,E1 -17190.729,E2 -17190.729} C_VEL
LIN {X 0,Y 289.061,Z 338.982,A -85,B 0,C 180,E1 -17191.393,E2 -17191.393} C_VEL
LIN {X 0,Y 289.552,Z 308.916,A -85,B 0,C 180,E1 -17192.138,E2 -17192.138} C_VEL
LIN {X 0,Y 286.634,Z 291.686,A -85,B 0,C 180,E1 -17192.735,E2 -17192.735} C_VEL
LIN {X 0,Y 284.771,Z 285.644,A -85,B 0,C 180,E1 -17193.006,E2 -17193.006} C_VEL
LIN {X 0,Y 284.597,Z 284.85,A -85,B 0,C 180,E1 -17193.363,E2 -17193.363} C_VEL
LIN {X 0,Y 284.653,Z 284.842,A -85,B 0,C 180,E1 -17197.091,E2 -17197.091} C_VEL
LIN {X 0,Y 284.487,Z 284.859,A -85,B 0,C 180,E1 -17199.958,E2 -17199.958} C_VEL
LIN {X 0,Y 284.438,Z 284.864,A -85,B 0,C 180,E1 -17204.305,E2 -17204.305} C_VEL
LIN {X 0,Y 284.372,Z 284.873,A -85,B 0,C 180,E1 -17208.741,E2 -17208.741} C_VEL
LIN {X 0,Y 284.302,Z 284.885,A -85,B 0,C 180,E1 -17213.299,E2 -17213.299} C_VEL
LIN {X 0,Y 284.301,Z 284.883,A -85,B 0,C 180,E1 -17217.15,E2 -17217.15} C_VEL
LIN {X 0,Y 284.269,Z 284.884,A -85,B 0,C 180,E1 -17220.095,E2 -17220.095} C_VEL
LIN {X 0,Y 284.278,Z 284.882,A -85,B 0,C 180,E1 -17222.949,E2 -17222.949} C_VEL
LIN {X 0,Y 284.293,Z 284.881,A -85,B 0,C 180,E1 -17226.392,E2 -17226.392} C_VEL
LIN {X 0,Y 284.259,Z 284.888,A -85,B 0,C 180,E1 -17230.003,E2 -17230.003} C_VEL
LIN {X 0,Y 284.213,Z 284.892,A -85,B 0,C 180,E1 -17234.192,E2 -17234.192} C_VEL
LIN {X 0,Y 284.253,Z 284.889,A -85,B 0,C 180,E1 -17238.129,E2 -17238.129} C_VEL
LIN {X 0,Y 284.311,Z 284.881,A -85,B 0,C 180,E1 -17242.282,E2 -17242.282} C_VEL
LIN {X 0,Y 284.294,Z 284.883,A -85,B 0,C 180,E1 -17245.356,E2 -17245.356} C_VEL
LIN {X 0,Y 284.272,Z 284.884,A -85,B 0,C 180,E1 -17248.729,E2 -17248.729} C_VEL
LIN {X 0,Y 284.272,Z 284.889,A -85,B 0,C 180,E1 -17251.989,E2 -17251.989} C_VEL
LIN {X 0,Y 284.314,Z 284.879,A -85,B 0,C 180,E1 -17256.151,E2 -17256.151} C_VEL
LIN {X 0,Y 284.415,Z 284.851,A -85,B 0,C 180,E1 -17260.926,E2 -17260.926} C_VEL
LIN {X 0,Y 284.556,Z 284.827,A -85,B 0,C 180,E1 -17262.487,E2 -17262.487} C_VEL
LIN {X 0,Y 286.663,Z 303.959,A -85,B 0,C 180,E1 -17263.272,E2 -17263.272} C_VEL
LIN {X 0,Y 286.921,Z 308.274,A -85,B 0,C 180,E1 -17263.441,E2 -17263.441} C_VEL
LIN {X 0,Y 286.878,Z 311.612,A -85,B 0,C 180,E1 -17263.568,E2 -17263.568} C_VEL
LIN {X 0,Y 286.129,Z 317.372,A -85,B 0,C 180,E1 -17263.78,E2 -17263.78} C_VEL
LIN {X 0,Y 279.798,Z 335.909,A -85,B 0,C 180,E1 -17264.441,E2 -17264.441} C_VEL
LIN {X 0,Y 279.03,Z 341.667,A -85,B 0,C 180,E1 -17264.664,E2 -17264.664} C_VEL
LIN {X 0,Y 278.506,Z 365.309,A -85,B 0,C 180,E1 -17265.669,E2 -17265.669} C_VEL
LIN {X 0,Y 278.136,Z 376.671,A -85,B 0,C 180,E1 -17266.395,E2 -17266.395} C_VEL
LIN {X 0,Y 277.691,Z 387.922,A -85,B 0,C 180,E1 -17267.397,E2 -17267.397} C_VEL
LIN {X 0,Y 277.264,Z 397.361,A -85,B 0,C 180,E1 -17268.491,E2 -17268.491} C_VEL
LIN {X 0,Y 276.762,Z 406.279,A -85,B 0,C 180,E1 -17269.766,E2 -17269.766} C_VEL
LIN {X 0,Y 276.252,Z 416.395,A -85,B 0,C 180,E1 -17271.593,E2 -17271.593} C_VEL
LIN {X 0,Y 275.915,Z 423.222,A -85,B 0,C 180,E1 -17273.139,E2 -17273.139} C_VEL
LIN {X 0,Y 275.674,Z 429.633,A -85,B 0,C 180,E1 -17274.908,E2 -17274.908} C_VEL
LIN {X 0,Y 275.595,Z 433.887,A -85,B 0,C 180,E1 -17276.35,E2 -17276.35} C_VEL
LIN {X 0,Y 275.358,Z 439.022,A -85,B 0,C 180,E1 -17278.542,E2 -17278.542} C_VEL
LIN {X 0,Y 275.356,Z 441.561,A -85,B 0,C 180,E1 -17280.005,E2 -17280.005} C_VEL
LIN {X 0,Y 275.459,Z 443.498,A -85,B 0,C 180,E1 -17281.467,E2 -17281.467} C_VEL
LIN {X 0,Y 275.699,Z 444.901,A -85,B 0,C 180,E1 -17282.927,E2 -17282.927} C_VEL
LIN {X 0,Y 276.105,Z 445.79,A -85,B 0,C 180,E1 -17284.384,E2 -17284.384} C_VEL
LIN {X 0,Y 276.577,Z 446.177,A -85,B 0,C 180,E1 -17285.838,E2 -17285.838} C_VEL
LIN {X 0,Y 277.034,Z 446.008,A -85,B 0,C 180,E1 -17287.292,E2 -17287.292} C_VEL
LIN {X 0,Y 277.616,Z 445.266,A -85,B 0,C 180,E1 -17288.741,E2 -17288.741} C_VEL
LIN {X 0,Y 279.339,Z 442.919,A -85,B 0,C 180,E1 -17291.121,E2 -17291.121} C_VEL
LIN {X 0,Y 280.939,Z 439.832,A -85,B 0,C 180,E1 -17293.016,E2 -17293.016} C_VEL
LIN {X 0,Y 283.057,Z 435.046,A -85,B 0,C 180,E1 -17295.116,E2 -17295.116} C_VEL
LIN {X 0,Y 285.158,Z 429.919,A -85,B 0,C 180,E1 -17296.838,E2 -17296.838} C_VEL
LIN {X 0,Y 287.999,Z 421.992,A -85,B 0,C 180,E1 -17298.869,E2 -17298.869} C_VEL
LIN {X 0,Y 290.056,Z 415.35,A -85,B 0,C 180,E1 -17300.203,E2 -17300.203} C_VEL
LIN {X 0,Y 292.564,Z 406.346,A -85,B 0,C 180,E1 -17301.679,E2 -17301.679} C_VEL
LIN {X 0,Y 294.98,Z 396.289,A -85,B 0,C 180,E1 -17302.967,E2 -17302.967} C_VEL
LIN {X 0,Y 296.877,Z 386.689,A -85,B 0,C 180,E1 -17303.92,E2 -17303.92} C_VEL
LIN {X 0,Y 298.495,Z 376.61,A -85,B 0,C 180,E1 -17304.707,E2 -17304.707} C_VEL
LIN {X 0,Y 300.229,Z 362.6,A -85,B 0,C 180,E1 -17305.462,E2 -17305.462} C_VEL
LIN {X 0,Y 303.886,Z 329.523,A -85,B 0,C 180,E1 -17306.904,E2 -17306.904} C_VEL
LIN {X 0,Y 300.453,Z 322.05,A -85,B 0,C 180,E1 -17308.304,E2 -17308.304} C_VEL
LIN {X 0,Y 296.398,Z 314.767,A -85,B 0,C 180,E1 -17310.063,E2 -17310.063} C_VEL
LIN {X 0,Y 293.762,Z 310.579,A -85,B 0,C 180,E1 -17311.311,E2 -17311.311} C_VEL
LIN {X 0,Y 291.687,Z 307.271,A -85,B 0,C 180,E1 -17312.431,E2 -17312.431} C_VEL
LIN {X 0,Y 288.632,Z 302.793,A -85,B 0,C 180,E1 -17314.269,E2 -17314.269} C_VEL
LIN {X 0,Y 285.481,Z 298.745,A -85,B 0,C 180,E1 -17316.573,E2 -17316.573} C_VEL
LIN {X 0,Y 282.414,Z 294.948,A -85,B 0,C 180,E1 -17319.838,E2 -17319.838} C_VEL
LIN {X 0,Y 280.869,Z 293.483,A -85,B 0,C 180,E1 -17322.952,E2 -17322.952} C_VEL
LIN {X 0,Y 281.154,Z 293.76,A -85,B 0,C 180,E1 -17326.466,E2 -17326.466} C_VEL
LIN {X 0,Y 282.36,Z 295.141,A -85,B 0,C 180,E1 -17329.409,E2 -17329.409} C_VEL
LIN {X 0,Y 285.86,Z 300.145,A -85,B 0,C 180,E1 -17333.152,E2 -17333.152} C_VEL
LIN {X 0,Y 289.588,Z 305.114,A -85,B 0,C 180,E1 -17335.704,E2 -17335.704} C_VEL
LIN {X 0,Y 293.653,Z 311.247,A -85,B 0,C 180,E1 -17337.962,E2 -17337.962} C_VEL
LIN {X 0,Y 297.315,Z 317.149,A -85,B 0,C 180,E1 -17339.684,E2 -17339.684} C_VEL
LIN {X 0,Y 298.948,Z 322.757,A -85,B 0,C 180,E1 -17340.623,E2 -17340.623} C_VEL
LIN {X 0,Y 300.311,Z 335.232,A -85,B 0,C 180,E1 -17341.942,E2 -17341.942} C_VEL
LIN {X 0,Y 301.217,Z 352.716,A -85,B 0,C 180,E1 -17343.394,E2 -17343.394} C_VEL
LIN {X 0,Y 301.029,Z 358.819,A -85,B 0,C 180,E1 -17343.769,E2 -17343.769} C_VEL
LIN {X 0,Y 297.462,Z 390.682,A -85,B 0,C 180,E1 -17345.205,E2 -17345.205} C_VEL
LIN {X 0,Y 295.367,Z 402.229,A -85,B 0,C 180,E1 -17345.953,E2 -17345.953} C_VEL
LIN {X 0,Y 293.037,Z 412.869,A -85,B 0,C 180,E1 -17346.875,E2 -17346.875} C_VEL
LIN {X 0,Y 290.287,Z 423.72,A -85,B 0,C 180,E1 -17348.146,E2 -17348.146} C_VEL
LIN {X 0,Y 287.741,Z 432.533,A -85,B 0,C 180,E1 -17349.445,E2 -17349.445} C_VEL
LIN {X 0,Y 285.245,Z 440.64,A -85,B 0,C 180,E1 -17350.946,E2 -17350.946} C_VEL
LIN {X 0,Y 282.838,Z 447.862,A -85,B 0,C 180,E1 -17352.652,E2 -17352.652} C_VEL
LIN {X 0,Y 280.786,Z 453.686,A -85,B 0,C 180,E1 -17354.391,E2 -17354.391} C_VEL
LIN {X 0,Y 279.071,Z 458.38,A -85,B 0,C 180,E1 -17356.158,E2 -17356.158} C_VEL
LIN {X 0,Y 277.477,Z 462.683,A -85,B 0,C 180,E1 -17358.309,E2 -17358.309} C_VEL
LIN {X 0,Y 276.684,Z 464.8,A -85,B 0,C 180,E1 -17359.758,E2 -17359.758} C_VEL
LIN {X 0,Y 276.046,Z 466.402,A -85,B 0,C 180,E1 -17361.213,E2 -17361.213} C_VEL
LIN {X 0,Y 275.632,Z 467.503,A -85,B 0,C 180,E1 -17362.675,E2 -17362.675} C_VEL
LIN {X 0,Y 275.391,Z 468.08,A -85,B 0,C 180,E1 -17364.46,E2 -17364.46} C_VEL
LIN {X 0,Y 275.4,Z 467.669,A -85,B 0,C 180,E1 -17367.074,E2 -17367.074} C_VEL
LIN {X 0,Y 275.393,Z 469.224,A -85,B 0,C 180,E1 -17368.537,E2 -17368.537} C_VEL
LIN {X 0,Y 275.414,Z 470.177,A -85,B 0,C 180,E1 -17370,E2 -17370} C_VEL
LIN {X 0,Y 275.347,Z 470.592,A -85,B 0,C 180,E1 -17371.462,E2 -17371.462} C_VEL
LIN {X 0,Y 275.372,Z 470.55,A -85,B 0,C 180,E1 -17372.926,E2 -17372.926} C_VEL
LIN {X 0,Y 275.316,Z 470.045,A -85,B 0,C 180,E1 -17374.392,E2 -17374.392} C_VEL
LIN {X 0,Y 275.392,Z 469.029,A -85,B 0,C 180,E1 -17375.859,E2 -17375.859} C_VEL
LIN {X 0,Y 275.763,Z 466.48,A -85,B 0,C 180,E1 -17378.057,E2 -17378.057} C_VEL
LIN {X 0,Y 276.499,Z 462.659,A -85,B 0,C 180,E1 -17380.249,E2 -17380.249} C_VEL
LIN {X 0,Y 277.626,Z 457.481,A -85,B 0,C 180,E1 -17382.426,E2 -17382.426} C_VEL
LIN {X 0,Y 278.841,Z 451.942,A -85,B 0,C 180,E1 -17384.225,E2 -17384.225} C_VEL
LIN {X 0,Y 280.405,Z 445.034,A -85,B 0,C 180,E1 -17386.004,E2 -17386.004} C_VEL
LIN {X 0,Y 282.344,Z 436.12,A -85,B 0,C 180,E1 -17387.753,E2 -17387.753} C_VEL
LIN {X 0,Y 283.73,Z 428.416,A -85,B 0,C 180,E1 -17388.972,E2 -17388.972} C_VEL
LIN {X 0,Y 284.98,Z 421.811,A -85,B 0,C 180,E1 -17389.821,E2 -17389.821} C_VEL
LIN {X 0,Y 286.168,Z 413.804,A -85,B 0,C 180,E1 -17390.673,E2 -17390.673} C_VEL
LIN {X 0,Y 287.375,Z 404.584,A -85,B 0,C 180,E1 -17391.426,E2 -17391.426} C_VEL
LIN {X 0,Y 288.369,Z 395.24,A -85,B 0,C 180,E1 -17391.982,E2 -17391.982} C_VEL
LIN {X 0,Y 289.059,Z 385.026,A -85,B 0,C 180,E1 -17392.389,E2 -17392.389} C_VEL
LIN {X 0,Y 289.858,Z 352.269,A -85,B 0,C 180,E1 -17393.247,E2 -17393.247} C_VEL
LIN {X 0,Y 287.342,Z 335.743,A -85,B 0,C 180,E1 -17393.987,E2 -17393.987} C_VEL
LIN {X 0,Y 283.735,Z 317.734,A -85,B 0,C 180,E1 -17394.914,E2 -17394.914} C_VEL
LIN {X 0,Y 281.753,Z 308.794,A -85,B 0,C 180,E1 -17395.447,E2 -17395.447} C_VEL
LIN {X 0,Y 281.533,Z 305.261,A -85,B 0,C 180,E1 -17396.701,E2 -17396.701} C_VEL
LIN {X 0,Y 279.729,Z 296.183,A -85,B 0,C 180,E1 -17400.164,E2 -17400.164} C_VEL
LIN {X 0,Y 277.289,Z 285.755,A -85,B 0,C 180,E1 -17404.466,E2 -17404.466} C_VEL
LIN {X 0,Y 277.263,Z 285.761,A -85,B 0,C 180,E1 -17408.202,E2 -17408.202} C_VEL
LIN {X 0,Y 277.224,Z 285.766,A -85,B 0,C 180,E1 -17412.672,E2 -17412.672} C_VEL
LIN {X 0,Y 277.201,Z 285.765,A -85,B 0,C 180,E1 -17416.796,E2 -17416.796} C_VEL
LIN {X 0,Y 277.205,Z 285.761,A -85,B 0,C 180,E1 -17420.663,E2 -17420.663} C_VEL
LIN {X 0,Y 277.287,Z 285.749,A -85,B 0,C 180,E1 -17424.338,E2 -17424.338} C_VEL
LIN {X 0,Y 277.248,Z 285.758,A -85,B 0,C 180,E1 -17427.833,E2 -17427.833} C_VEL
LIN {X 0,Y 277.251,Z 285.761,A -85,B 0,C 180,E1 -17431.204,E2 -17431.204} C_VEL
LIN {X 0,Y 277.261,Z 285.755,A -85,B 0,C 180,E1 -17434.47,E2 -17434.47} C_VEL
LIN {X 0,Y 277.271,Z 285.752,A -85,B 0,C 180,E1 -17437.649,E2 -17437.649} C_VEL
LIN {X 0,Y 277.33,Z 285.749,A -85,B 0,C 180,E1 -17440.761,E2 -17440.761} C_VEL
LIN {X 0,Y 277.414,Z 285.734,A -85,B 0,C 180,E1 -17445.321,E2 -17445.321} C_VEL
LIN {X 0,Y 277.465,Z 285.72,A -85,B 0,C 180,E1 -17449.783,E2 -17449.783} C_VEL
LIN {X 0,Y 277.644,Z 285.704,A -85,B 0,C 180,E1 -17452.724,E2 -17452.724} C_VEL
LIN {X 0,Y 277.817,Z 285.68,A -85,B 0,C 180,E1 -17458.546,E2 -17458.546} C_VEL
LIN {X 0,Y 277.817,Z 285.682,A -85,B 0,C 180,E1 -17461.445,E2 -17461.445} C_VEL
LIN {X 0,Y 277.608,Z 285.713,A -85,B 0,C 180,E1 -17467.267,E2 -17467.267} C_VEL
LIN {X 0,Y 277.453,Z 285.726,A -85,B 0,C 180,E1 -17470.208,E2 -17470.208} C_VEL
LIN {X 0,Y 277.428,Z 285.733,A -85,B 0,C 180,E1 -17474.669,E2 -17474.669} C_VEL
LIN {X 0,Y 277.336,Z 285.747,A -85,B 0,C 180,E1 -17479.229,E2 -17479.229} C_VEL
LIN {X 0,Y 277.308,Z 285.749,A -85,B 0,C 180,E1 -17484.165,E2 -17484.165} C_VEL
LIN {X 0,Y 277.311,Z 285.752,A -85,B 0,C 180,E1 -17487.5,E2 -17487.5} C_VEL
LIN {X 0,Y 277.258,Z 285.762,A -85,B 0,C 180,E1 -17490.476,E2 -17490.476} C_VEL
LIN {X 0,Y 277.23,Z 285.765,A -85,B 0,C 180,E1 -17493.891,E2 -17493.891} C_VEL
LIN {X 0,Y 277.26,Z 285.756,A -85,B 0,C 180,E1 -17497.463,E2 -17497.463} C_VEL
LIN {X 0,Y 277.248,Z 285.755,A -85,B 0,C 180,E1 -17501.221,E2 -17501.221} C_VEL
LIN {X 0,Y 277.267,Z 285.759,A -85,B 0,C 180,E1 -17505.204,E2 -17505.204} C_VEL
LIN {X 0,Y 277.317,Z 285.787,A -85,B 0,C 180,E1 -17506.57,E2 -17506.57} C_VEL
LIN {X 0,Y 277.647,Z 287.152,A -85,B 0,C 180,E1 -17507.113,E2 -17507.113} C_VEL
LIN {X 0,Y 286.799,Z 306.262,A -85,B 0,C 180,E1 -17508.783,E2 -17508.783} C_VEL
LIN {X 0,Y 291.002,Z 316.634,A -85,B 0,C 180,E1 -17509.548,E2 -17509.548} C_VEL
LIN {X 0,Y 289.58,Z 363.68,A -85,B 0,C 180,E1 -17510.769,E2 -17510.769} C_VEL
LIN {X 0,Y 288.987,Z 373.563,A -85,B 0,C 180,E1 -17511.217,E2 -17511.217} C_VEL
LIN {X 0,Y 288.019,Z 384.999,A -85,B 0,C 180,E1 -17512.007,E2 -17512.007} C_VEL
LIN {X 0,Y 286.828,Z 394.195,A -85,B 0,C 180,E1 -17512.888,E2 -17512.888} C_VEL
LIN {X 0,Y 285.494,Z 403.313,A -85,B 0,C 180,E1 -17514.029,E2 -17514.029} C_VEL
LIN {X 0,Y 284.295,Z 410.145,A -85,B 0,C 180,E1 -17515.076,E2 -17515.076} C_VEL
LIN {X 0,Y 282.813,Z 417.414,A -85,B 0,C 180,E1 -17516.433,E2 -17516.433} C_VEL
LIN {X 0,Y 281.72,Z 422.474,A -85,B 0,C 180,E1 -17517.565,E2 -17517.565} C_VEL
LIN {X 0,Y 280.397,Z 428.099,A -85,B 0,C 180,E1 -17519.082,E2 -17519.082} C_VEL
LIN {X 0,Y 279.3,Z 432.74,A -85,B 0,C 180,E1 -17520.615,E2 -17520.615} C_VEL
LIN {X 0,Y 278.365,Z 436.373,A -85,B 0,C 180,E1 -17522.073,E2 -17522.073} C_VEL
LIN {X 0,Y 277.493,Z 439.59,A -85,B 0,C 180,E1 -17523.691,E2 -17523.691} C_VEL
LIN {X 0,Y 276.832,Z 441.96,A -85,B 0,C 180,E1 -17525.236,E2 -17525.236} C_VEL
LIN {X 0,Y 276.043,Z 444.281,A -85,B 0,C 180,E1 -17527.549,E2 -17527.549} C_VEL
LIN {X 0,Y 275.651,Z 445.191,A -85,B 0,C 180,E1 -17529.088,E2 -17529.088} C_VEL
LIN {X 0,Y 275.385,Z 445.513,A -85,B 0,C 180,E1 -17530.76,E2 -17530.76} C_VEL
LIN {X 0,Y 275.258,Z 445.223,A -85,B 0,C 180,E1 -17532.159,E2 -17532.159} C_VEL
LIN {X 0,Y 275.229,Z 444.436,A -85,B 0,C 180,E1 -17533.687,E2 -17533.687} C_VEL
LIN {X 0,Y 275.344,Z 442.374,A -85,B 0,C 180,E1 -17535.885,E2 -17535.885} C_VEL
LIN {X 0,Y 275.691,Z 438.854,A -85,B 0,C 180,E1 -17538.233,E2 -17538.233} C_VEL
LIN {X 0,Y 276.155,Z 433.876,A -85,B 0,C 180,E1 -17540.479,E2 -17540.479} C_VEL
LIN {X 0,Y 276.666,Z 429.187,A -85,B 0,C 180,E1 -17542.128,E2 -17542.128} C_VEL
LIN {X 0,Y 277.182,Z 423.257,A -85,B 0,C 180,E1 -17543.814,E2 -17543.814} C_VEL
LIN {X 0,Y 277.875,Z 416.894,A -85,B 0,C 180,E1 -17545.285,E2 -17545.285} C_VEL
LIN {X 0,Y 278.647,Z 409.164,A -85,B 0,C 180,E1 -17546.747,E2 -17546.747} C_VEL
LIN {X 0,Y 279.623,Z 399.489,A -85,B 0,C 180,E1 -17548.2,E2 -17548.2} C_VEL
LIN {X 0,Y 280.407,Z 389.984,A -85,B 0,C 180,E1 -17549.282,E2 -17549.282} C_VEL
LIN {X 0,Y 280.961,Z 380.922,A -85,B 0,C 180,E1 -17550.082,E2 -17550.082} C_VEL
LIN {X 0,Y 281.429,Z 371.253,A -85,B 0,C 180,E1 -17550.712,E2 -17550.712} C_VEL
LIN {X 0,Y 281.687,Z 361.96,A -85,B 0,C 180,E1 -17551.123,E2 -17551.123} C_VEL
LIN {X 0,Y 282.68,Z 309.73,A -85,B 0,C 180,E1 -17552.478,E2 -17552.478} C_VEL
LIN {X 0,Y 279.961,Z 293.551,A -85,B 0,C 180,E1 -17553.055,E2 -17553.055} C_VEL
LIN {X 0,Y 277.585,Z 285.976,A -85,B 0,C 180,E1 -17553.402,E2 -17553.402} C_VEL
LIN {X 0,Y 277.532,Z 285.729,A -85,B 0,C 180,E1 -17553.63,E2 -17553.63} C_VEL
LIN {X 0,Y 277.608,Z 285.719,A -85,B 0,C 180,E1 -17557.272,E2 -17557.272} C_VEL
LIN {X 0,Y 277.429,Z 285.738,A -85,B 0,C 180,E1 -17560.214,E2 -17560.214} C_VEL
LIN {X 0,Y 277.384,Z 285.744,A -85,B 0,C 180,E1 -17564.677,E2 -17564.677} C_VEL
LIN {X 0,Y 277.314,Z 285.755,A -85,B 0,C 180,E1 -17569.236,E2 -17569.236} C_VEL
LIN {X 0,Y 277.256,Z 285.76,A -85,B 0,C 180,E1 -17573.928,E2 -17573.928} C_VEL
LIN {X 0,Y 277.242,Z 285.765,A -85,B 0,C 180,E1 -17577.486,E2 -17577.486} C_VEL
LIN {X 0,Y 277.222,Z 285.761,A -85,B 0,C 180,E1 -17580.476,E2 -17580.476} C_VEL
LIN {X 0,Y 277.22,Z 285.764,A -85,B 0,C 180,E1 -17583.9,E2 -17583.9} C_VEL
LIN {X 0,Y 277.227,Z 285.765,A -85,B 0,C 180,E1 -17587.476,E2 -17587.476} C_VEL
LIN {X 0,Y 277.161,Z 285.771,A -85,B 0,C 180,E1 -17591.246,E2 -17591.246} C_VEL
LIN {X 0,Y 277.178,Z 285.768,A -85,B 0,C 180,E1 -17595.232,E2 -17595.232} C_VEL
LIN {X 0,Y 277.205,Z 285.767,A -85,B 0,C 180,E1 -17599.517,E2 -17599.517} C_VEL
LIN {X 0,Y 277.255,Z 285.759,A -85,B 0,C 180,E1 -17602.536,E2 -17602.536} C_VEL
LIN {X 0,Y 277.232,Z 285.763,A -85,B 0,C 180,E1 -17606.109,E2 -17606.109} C_VEL
LIN {X 0,Y 277.249,Z 285.76,A -85,B 0,C 180,E1 -17609.544,E2 -17609.544} C_VEL
LIN {X 0,Y 277.281,Z 285.755,A -85,B 0,C 180,E1 -17612.862,E2 -17612.862} C_VEL
LIN {X 0,Y 277.275,Z 285.756,A -85,B 0,C 180,E1 -17616.081,E2 -17616.081} C_VEL
LIN {X 0,Y 277.367,Z 285.734,A -85,B 0,C 180,E1 -17620.773,E2 -17620.773} C_VEL
LIN {X 0,Y 277.532,Z 285.702,A -85,B 0,C 180,E1 -17622.389,E2 -17622.389} C_VEL
LIN {X 0,Y 279.846,Z 308.201,A -85,B 0,C 180,E1 -17623.333,E2 -17623.333} C_VEL
LIN {X 0,Y 279.03,Z 341.667,A -85,B 0,C 180,E1 -17624.664,E2 -17624.664} C_VEL
LIN {X 0,Y 278.278,Z 347.429,A -85,B 0,C 180,E1 -17624.888,E2 -17624.888} C_VEL
LIN {X 0,Y 272.016,Z 365.873,A -85,B 0,C 180,E1 -17625.699,E2 -17625.699} C_VEL
LIN {X 0,Y 271.229,Z 371.505,A -85,B 0,C 180,E1 -17626.041,E2 -17626.041} C_VEL
LIN {X 0,Y 270.777,Z 383.154,A -85,B 0,C 180,E1 -17626.974,E2 -17626.974} C_VEL
LIN {X 0,Y 270.301,Z 394.641,A -85,B 0,C 180,E1 -17628.19,E2 -17628.19} C_VEL
LIN {X 0,Y 269.779,Z 404.047,A -85,B 0,C 180,E1 -17629.498,E2 -17629.498} C_VEL
LIN {X 0,Y 269.324,Z 412.83,A -85,B 0,C 180,E1 -17630.997,E2 -17630.997} C_VEL
LIN {X 0,Y 268.888,Z 421.667,A -85,B 0,C 180,E1 -17632.874,E2 -17632.874} C_VEL
LIN {X 0,Y 268.581,Z 427.449,A -85,B 0,C 180,E1 -17634.416,E2 -17634.416} C_VEL
LIN {X 0,Y 268.539,Z 433.082,A -85,B 0,C 180,E1 -17636.254,E2 -17636.254} C_VEL
LIN {X 0,Y 268.284,Z 438.466,A -85,B 0,C 180,E1 -17638.504,E2 -17638.504} C_VEL
LIN {X 0,Y 268.306,Z 442.423,A -85,B 0,C 180,E1 -17640.755,E2 -17640.755} C_VEL
LIN {X 0,Y 268.63,Z 444.962,A -85,B 0,C 180,E1 -17643.004,E2 -17643.004} C_VEL
LIN {X 0,Y 269.048,Z 446.043,A -85,B 0,C 180,E1 -17644.499,E2 -17644.499} C_VEL
LIN {X 0,Y 269.536,Z 446.546,A -85,B 0,C 180,E1 -17645.991,E2 -17645.991} C_VEL
LIN {X 0,Y 270.026,Z 446.489,A -85,B 0,C 180,E1 -17647.482,E2 -17647.482} C_VEL
LIN {X 0,Y 270.66,Z 445.95,A -85,B 0,C 180,E1 -17648.968,E2 -17648.968} C_VEL
LIN {X 0,Y 271.815,Z 444.871,A -85,B 0,C 180,E1 -17650.432,E2 -17650.432} C_VEL
LIN {X 0,Y 272.813,Z 443.308,A -85,B 0,C 180,E1 -17651.898,E2 -17651.898} C_VEL
LIN {X 0,Y 274.859,Z 439.779,A -85,B 0,C 180,E1 -17654.063,E2 -17654.063} C_VEL
LIN {X 0,Y 277.255,Z 434.896,A -85,B 0,C 180,E1 -17656.195,E2 -17656.195} C_VEL
LIN {X 0,Y 280.034,Z 428.394,A -85,B 0,C 180,E1 -17658.287,E2 -17658.287} C_VEL
LIN {X 0,Y 282.64,Z 421.457,A -85,B 0,C 180,E1 -17659.997,E2 -17659.997} C_VEL
LIN {X 0,Y 284.904,Z 414.732,A -85,B 0,C 180,E1 -17661.341,E2 -17661.341} C_VEL
LIN {X 0,Y 287.632,Z 405.529,A -85,B 0,C 180,E1 -17662.827,E2 -17662.827} C_VEL
LIN {X 0,Y 290.155,Z 395.035,A -85,B 0,C 180,E1 -17664.13,E2 -17664.13} C_VEL
LIN {X 0,Y 292.603,Z 383.455,A -85,B 0,C 180,E1 -17665.239,E2 -17665.239} C_VEL
LIN {X 0,Y 294.392,Z 372.06,A -85,B 0,C 180,E1 -17666.023,E2 -17666.023} C_VEL
LIN {X 0,Y 296.303,Z 356.806,A -85,B 0,C 180,E1 -17666.742,E2 -17666.742} C_VEL
LIN {X 0,Y 299.113,Z 332.629,A -85,B 0,C 180,E1 -17667.834,E2 -17667.834} C_VEL
LIN {X 0,Y 295.701,Z 325.114,A -85,B 0,C 180,E1 -17669.367,E2 -17669.367} C_VEL
LIN {X 0,Y 291.577,Z 317.677,A -85,B 0,C 180,E1 -17671.383,E2 -17671.383} C_VEL
LIN {X 0,Y 288.625,Z 313.077,A -85,B 0,C 180,E1 -17673.013,E2 -17673.013} C_VEL
LIN {X 0,Y 286.288,Z 309.341,A -85,B 0,C 180,E1 -17674.551,E2 -17674.551} C_VEL
LIN {X 0,Y 283.015,Z 304.961,A -85,B 0,C 180,E1 -17677.108,E2 -17677.108} C_VEL
LIN {X 0,Y 280.251,Z 301.49,A -85,B 0,C 180,E1 -17680.438,E2 -17680.438} C_VEL
LIN {X 0,Y 279.115,Z 300.333,A -85,B 0,C 180,E1 -17683.096,E2 -17683.096} C_VEL
LIN {X 0,Y 279.158,Z 300.55,A -85,B 0,C 180,E1 -17686.411,E2 -17686.411} C_VEL
LIN {X 0,Y 280.465,Z 301.931,A -85,B 0,C 180,E1 -17689.22,E2 -17689.22} C_VEL
LIN {X 0,Y 283.864,Z 307.076,A -85,B 0,C 180,E1 -17693.038,E2 -17693.038} C_VEL
LIN {X 0,Y 287.067,Z 311.562,A -85,B 0,C 180,E1 -17695.351,E2 -17695.351} C_VEL
LIN {X 0,Y 290.787,Z 317.375,A -85,B 0,C 180,E1 -17697.538,E2 -17697.538} C_VEL
LIN {X 0,Y 293.902,Z 322.703,A -85,B 0,C 180,E1 -17699.121,E2 -17699.121} C_VEL
LIN {X 0,Y 295.045,Z 327.992,A -85,B 0,C 180,E1 -17699.939,E2 -17699.939} C_VEL
LIN {X 0,Y 295.969,Z 339.151,A -85,B 0,C 180,E1 -17701.121,E2 -17701.121} C_VEL
LIN {X 0,Y 296.465,Z 355.631,A -85,B 0,C 180,E1 -17702.523,E2 -17702.523} C_VEL
LIN {X 0,Y 296.258,Z 359.86,A -85,B 0,C 180,E1 -17702.776,E2 -17702.776} C_VEL
LIN {X 0,Y 292.704,Z 389.647,A -85,B 0,C 180,E1 -17704.148,E2 -17704.148} C_VEL
LIN {X 0,Y 290.374,Z 401.727,A -85,B 0,C 180,E1 -17704.94,E2 -17704.94} C_VEL
LIN {X 0,Y 287.509,Z 413.899,A -85,B 0,C 180,E1 -17706.021,E2 -17706.021} C_VEL
LIN {X 0,Y 284.599,Z 424.396,A -85,B 0,C 180,E1 -17707.303,E2 -17707.303} C_VEL
LIN {X 0,Y 282.24,Z 431.946,A -85,B 0,C 180,E1 -17708.451,E2 -17708.451} C_VEL
LIN {X 0,Y 279.243,Z 440.829,A -85,B 0,C 180,E1 -17710.137,E2 -17710.137} C_VEL
LIN {X 0,Y 276.64,Z 447.908,A -85,B 0,C 180,E1 -17711.868,E2 -17711.868} C_VEL
LIN {X 0,Y 274.46,Z 453.619,A -85,B 0,C 180,E1 -17713.64,E2 -17713.64} C_VEL
LIN {X 0,Y 272.85,Z 457.401,A -85,B 0,C 180,E1 -17715.073,E2 -17715.073} C_VEL
LIN {X 0,Y 271.035,Z 461.824,A -85,B 0,C 180,E1 -17717.267,E2 -17717.267} C_VEL
LIN {X 0,Y 269.687,Z 464.981,A -85,B 0,C 180,E1 -17719.489,E2 -17719.489} C_VEL
LIN {X 0,Y 269.033,Z 466.355,A -85,B 0,C 180,E1 -17720.982,E2 -17720.982} C_VEL
LIN {X 0,Y 268.573,Z 467.246,A -85,B 0,C 180,E1 -17722.482,E2 -17722.482} C_VEL
LIN {X 0,Y 268.312,Z 467.609,A -85,B 0,C 180,E1 -17724.499,E2 -17724.499} C_VEL
LIN {X 0,Y 268.331,Z 466.974,A -85,B 0,C 180,E1 -17726.621,E2 -17726.621} C_VEL
LIN {X 0,Y 268.314,Z 468.791,A -85,B 0,C 180,E1 -17728.499,E2 -17728.499} C_VEL
LIN {X 0,Y 268.332,Z 469.765,A -85,B 0,C 180,E1 -17730,E2 -17730} C_VEL
LIN {X 0,Y 268.271,Z 470.237,A -85,B 0,C 180,E1 -17731.501,E2 -17731.501} C_VEL
LIN {X 0,Y 268.277,Z 470.248,A -85,B 0,C 180,E1 -17733.003,E2 -17733.003} C_VEL
LIN {X 0,Y 268.23,Z 469.798,A -85,B 0,C 180,E1 -17734.508,E2 -17734.508} C_VEL
LIN {X 0,Y 268.316,Z 468.79,A -85,B 0,C 180,E1 -17736.014,E2 -17736.014} C_VEL
LIN {X 0,Y 268.723,Z 466.343,A -85,B 0,C 180,E1 -17738.27,E2 -17738.27} C_VEL
LIN {X 0,Y 269.513,Z 462.591,A -85,B 0,C 180,E1 -17740.517,E2 -17740.517} C_VEL
LIN {X 0,Y 270.234,Z 459.411,A -85,B 0,C 180,E1 -17742.008,E2 -17742.008} C_VEL
LIN {X 0,Y 271.457,Z 454.382,A -85,B 0,C 180,E1 -17743.856,E2 -17743.856} C_VEL
LIN {X 0,Y 272.887,Z 448.09,A -85,B 0,C 180,E1 -17745.689,E2 -17745.689} C_VEL
LIN {X 0,Y 274.351,Z 441.949,A -85,B 0,C 180,E1 -17747.133,E2 -17747.133} C_VEL
LIN {X 0,Y 275.798,Z 435.519,A -85,B 0,C 180,E1 -17748.381,E2 -17748.381} C_VEL
LIN {X 0,Y 277.045,Z 428.988,A -85,B 0,C 180,E1 -17749.448,E2 -17749.448} C_VEL
LIN {X 0,Y 278.582,Z 421.087,A -85,B 0,C 180,E1 -17750.489,E2 -17750.489} C_VEL
LIN {X 0,Y 279.809,Z 412.988,A -85,B 0,C 180,E1 -17751.358,E2 -17751.358} C_VEL
LIN {X 0,Y 281.102,Z 403.779,A -85,B 0,C 180,E1 -17752.109,E2 -17752.109} C_VEL
LIN {X 0,Y 282.146,Z 394.418,A -85,B 0,C 180,E1 -17752.664,E2 -17752.664} C_VEL
LIN {X 0,Y 282.822,Z 383.947,A -85,B 0,C 180,E1 -17753.081,E2 -17753.081} C_VEL
LIN {X 0,Y 283.659,Z 353.608,A -85,B 0,C 180,E1 -17753.88,E2 -17753.88} C_VEL
LIN {X 0,Y 281.277,Z 337.709,A -85,B 0,C 180,E1 -17754.613,E2 -17754.613} C_VEL
LIN {X 0,Y 277.921,Z 320.467,A -85,B 0,C 180,E1 -17755.523,E2 -17755.523} C_VEL
LIN {X 0,Y 275.303,Z 310.001,A -85,B 0,C 180,E1 -17756.165,E2 -17756.165} C_VEL
LIN {X 0,Y 274.907,Z 308.4,A -85,B 0,C 180,E1 -17756.305,E2 -17756.305} C_VEL
LIN {X 0,Y 273.268,Z 299.712,A -85,B 0,C 180,E1 -17759.675,E2 -17759.675} C_VEL
LIN {X 0,Y 270.943,Z 289.586,A -85,B 0,C 180,E1 -17763.891,E2 -17763.891} C_VEL
LIN {X 0,Y 270.234,Z 286.625,A -85,B 0,C 180,E1 -17765.242,E2 -17765.242} C_VEL
LIN {X 0,Y 270.209,Z 286.637,A -85,B 0,C 180,E1 -17768.708,E2 -17768.708} C_VEL
LIN {X 0,Y 270.175,Z 286.643,A -85,B 0,C 180,E1 -17773.246,E2 -17773.246} C_VEL
LIN {X 0,Y 270.16,Z 286.64,A -85,B 0,C 180,E1 -17777.435,E2 -17777.435} C_VEL
LIN {X 0,Y 270.174,Z 286.636,A -85,B 0,C 180,E1 -17781.364,E2 -17781.364} C_VEL
LIN {X 0,Y 270.207,Z 286.63,A -85,B 0,C 180,E1 -17785.091,E2 -17785.091} C_VEL
LIN {X 0,Y 270.192,Z 286.631,A -85,B 0,C 180,E1 -17789.133,E2 -17789.133} C_VEL
LIN {X 0,Y 270.231,Z 286.633,A -85,B 0,C 180,E1 -17792.159,E2 -17792.159} C_VEL
LIN {X 0,Y 270.236,Z 286.634,A -85,B 0,C 180,E1 -17795.538,E2 -17795.538} C_VEL
LIN {X 0,Y 270.283,Z 286.628,A -85,B 0,C 180,E1 -17800.239,E2 -17800.239} C_VEL
LIN {X 0,Y 270.382,Z 286.609,A -85,B 0,C 180,E1 -17804.93,E2 -17804.93} C_VEL
LIN {X 0,Y 270.417,Z 286.596,A -85,B 0,C 180,E1 -17809.514,E2 -17809.514} C_VEL
LIN {X 0,Y 270.602,Z 286.582,A -85,B 0,C 180,E1 -17812.534,E2 -17812.534} C_VEL
LIN {X 0,Y 270.783,Z 286.557,A -85,B 0,C 180,E1 -17818.508,E2 -17818.508} C_VEL
LIN {X 0,Y 270.783,Z 286.559,A -85,B 0,C 180,E1 -17821.482,E2 -17821.482} C_VEL
LIN {X 0,Y 270.567,Z 286.591,A -85,B 0,C 180,E1 -17827.457,E2 -17827.457} C_VEL
LIN {X 0,Y 270.405,Z 286.603,A -85,B 0,C 180,E1 -17830.477,E2 -17830.477} C_VEL
LIN {X 0,Y 270.396,Z 286.607,A -85,B 0,C 180,E1 -17835.059,E2 -17835.059} C_VEL
LIN {X 0,Y 270.293,Z 286.622,A -85,B 0,C 180,E1 -17839.75,E2 -17839.75} C_VEL
LIN {X 0,Y 270.263,Z 286.625,A -85,B 0,C 180,E1 -17844.58,E2 -17844.58} C_VEL
LIN {X 0,Y 270.257,Z 286.629,A -85,B 0,C 180,E1 -17847.904,E2 -17847.904} C_VEL
LIN {X 0,Y 270.169,Z 286.64,A -85,B 0,C 180,E1 -17851.343,E2 -17851.343} C_VEL
LIN {X 0,Y 270.186,Z 286.629,A -85,B 0,C 180,E1 -17854.9,E2 -17854.9} C_VEL
LIN {X 0,Y 270.204,Z 286.64,A -85,B 0,C 180,E1 -17858.712,E2 -17858.712} C_VEL
LIN {X 0,Y 270.238,Z 286.639,A -85,B 0,C 180,E1 -17862.537,E2 -17862.537} C_VEL
LIN {X 0,Y 270.276,Z 286.779,A -85,B 0,C 180,E1 -17865.886,E2 -17865.886} C_VEL
LIN {X 0,Y 270.443,Z 287.565,A -85,B 0,C 180,E1 -17866.176,E2 -17866.176} C_VEL
LIN {X 0,Y 272.283,Z 291.092,A -85,B 0,C 180,E1 -17866.534,E2 -17866.534} C_VEL
LIN {X 0,Y 280.059,Z 307.152,A -85,B 0,C 180,E1 -17868.015,E2 -17868.015} C_VEL
LIN {X 0,Y 284.806,Z 318.586,A -85,B 0,C 180,E1 -17868.911,E2 -17868.911} C_VEL
LIN {X 0,Y 283.297,Z 364.171,A -85,B 0,C 180,E1 -17870.113,E2 -17870.113} C_VEL
LIN {X 0,Y 282.662,Z 374.615,A -85,B 0,C 180,E1 -17870.606,E2 -17870.606} C_VEL
LIN {X 0,Y 281.503,Z 386.68,A -85,B 0,C 180,E1 -17871.495,E2 -17871.495} C_VEL
LIN {X 0,Y 280.349,Z 395.088,A -85,B 0,C 180,E1 -17872.335,E2 -17872.335} C_VEL
LIN {X 0,Y 278.985,Z 403.88,A -85,B 0,C 180,E1 -17873.465,E2 -17873.465} C_VEL
LIN {X 0,Y 277.653,Z 411.147,A -85,B 0,C 180,E1 -17874.619,E2 -17874.619} C_VEL
LIN {X 0,Y 276.149,Z 418.059,A -85,B 0,C 180,E1 -17875.951,E2 -17875.951} C_VEL
LIN {X 0,Y 274.647,Z 424.558,A -85,B 0,C 180,E1 -17877.495,E2 -17877.495} C_VEL
LIN {X 0,Y 273.008,Z 431.114,A -85,B 0,C 180,E1 -17879.442,E2 -17879.442} C_VEL
LIN {X 0,Y 271.537,Z 436.649,A -85,B 0,C 180,E1 -17881.628,E2 -17881.628} C_VEL
LIN {X 0,Y 270.375,Z 440.618,A -85,B 0,C 180,E1 -17883.776,E2 -17883.776} C_VEL
LIN {X 0,Y 269.468,Z 443.361,A -85,B 0,C 180,E1 -17885.884,E2 -17885.884} C_VEL
LIN {X 0,Y 269.135,Z 444.403,A -85,B 0,C 180,E1 -17886.94,E2 -17886.94} C_VEL
LIN {X 0,Y 268.686,Z 445.382,A -85,B 0,C 180,E1 -17888.519,E2 -17888.519} C_VEL
LIN {X 0,Y 268.359,Z 445.837,A -85,B 0,C 180,E1 -17890.506,E2 -17890.506} C_VEL
LIN {X 0,Y 268.143,Z 444.983,A -85,B 0,C 180,E1 -17893.244,E2 -17893.244} C_VEL
LIN {X 0,Y 268.176,Z 443.819,A -85,B 0,C 180,E1 -17894.808,E2 -17894.808} C_VEL
LIN {X 0,Y 268.322,Z 442.093,A -85,B 0,C 180,E1 -17896.366,E2 -17896.366} C_VEL
LIN {X 0,Y 268.666,Z 438.295,A -85,B 0,C 180,E1 -17898.686,E2 -17898.686} C_VEL
LIN {X 0,Y 268.998,Z 435.031,A -85,B 0,C 180,E1 -17900.223,E2 -17900.223} C_VEL
LIN {X 0,Y 269.572,Z 429.86,A -85,B 0,C 180,E1 -17902.128,E2 -17902.128} C_VEL
LIN {X 0,Y 270.018,Z 424.8,A -85,B 0,C 180,E1 -17903.649,E2 -17903.649} C_VEL
LIN {X 0,Y 270.713,Z 418.676,A -85,B 0,C 180,E1 -17905.16,E2 -17905.16} C_VEL
LIN {X 0,Y 271.486,Z 411.229,A -85,B 0,C 180,E1 -17906.661,E2 -17906.661} C_VEL
LIN {X 0,Y 272.292,Z 403.249,A -85,B 0,C 180,E1 -17907.966,E2 -17907.966} C_VEL
LIN {X 0,Y 273.095,Z 394.792,A -85,B 0,C 180,E1 -17909.079,E2 -17909.079} C_VEL
LIN {X 0,Y 273.936,Z 383.539,A -85,B 0,C 180,E1 -17910.218,E2 -17910.218} C_VEL
LIN {X 0,Y 274.474,Z 373.07,A -85,B 0,C 180,E1 -17910.956,E2 -17910.956} C_VEL
LIN {X 0,Y 274.775,Z 363.541,A -85,B 0,C 180,E1 -17911.415,E2 -17911.415} C_VEL
LIN {X 0,Y 275.777,Z 317.327,A -85,B 0,C 180,E1 -17912.654,E2 -17912.654} C_VEL
LIN {X 0,Y 275.759,Z 310.113,A -85,B 0,C 180,E1 -17912.849,E2 -17912.849} C_VEL
LIN {X 0,Y 273.324,Z 295.488,A -85,B 0,C 180,E1 -17913.386,E2 -17913.386} C_VEL
LIN {X 0,Y 270.479,Z 286.607,A -85,B 0,C 180,E1 -17913.818,E2 -17913.818} C_VEL
LIN {X 0,Y 270.566,Z 286.594,A -85,B 0,C 180,E1 -17917.463,E2 -17917.463} C_VEL
LIN {X 0,Y 270.381,Z 286.616,A -85,B 0,C 180,E1 -17920.484,E2 -17920.484} C_VEL
LIN {X 0,Y 270.352,Z 286.622,A -85,B 0,C 180,E1 -17925.068,E2 -17925.068} C_VEL
LIN {X 0,Y 270.272,Z 286.63,A -85,B 0,C 180,E1 -17929.758,E2 -17929.758} C_VEL
LIN {X 0,Y 270.197,Z 286.639,A -85,B 0,C 180,E1 -17934.593,E2 -17934.593} C_VEL
LIN {X 0,Y 270.171,Z 286.643,A -85,B 0,C 180,E1 -17937.92,E2 -17937.92} C_VEL
LIN {X 0,Y 270.147,Z 286.644,A -85,B 0,C 180,E1 -17941.353,E2 -17941.353} C_VEL
LIN {X 0,Y 270.172,Z 286.64,A -85,B 0,C 180,E1 -17944.91,E2 -17944.91} C_VEL
LIN {X 0,Y 270.175,Z 286.639,A -85,B 0,C 180,E1 -17948.715,E2 -17948.715} C_VEL
LIN {X 0,Y 270.127,Z 286.647,A -85,B 0,C 180,E1 -17953.249,E2 -17953.249} C_VEL
LIN {X 0,Y 270.153,Z 286.646,A -85,B 0,C 180,E1 -17957.447,E2 -17957.447} C_VEL
LIN {X 0,Y 270.191,Z 286.638,A -85,B 0,C 180,E1 -17961.379,E2 -17961.379} C_VEL
LIN {X 0,Y 270.187,Z 286.639,A -85,B 0,C 180,E1 -17965.1,E2 -17965.1} C_VEL
LIN {X 0,Y 270.171,Z 286.64,A -85,B 0,C 180,E1 -17969.142,E2 -17969.142} C_VEL
LIN {X 0,Y 270.211,Z 286.639,A -85,B 0,C 180,E1 -17972.168,E2 -17972.168} C_VEL
LIN {X 0,Y 270.219,Z 286.634,A -85,B 0,C 180,E1 -17975.548,E2 -17975.548} C_VEL
LIN {X 0,Y 270.308,Z 286.621,A -85,B 0,C 180,E1 -17980.251,E2 -17980.251} C_VEL
LIN {X 0,Y 270.46,Z 286.583,A -85,B 0,C 180,E1 -17982.284,E2 -17982.284} C_VEL
LIN {X 0,Y 272.774,Z 308.808,A -85,B 0,C 180,E1 -17983.275,E2 -17983.275} C_VEL
LIN {X 0,Y 271.41,Z 365.169,A -85,B 0,C 180,E1 -17985.669,E2 -17985.669} C_VEL
LIN {X 0,Y 271.229,Z 371.505,A -85,B 0,C 180,E1 -17986.041,E2 -17986.041} C_VEL
LIN {X 0,Y 270.437,Z 377.04,A -85,B 0,C 180,E1 -17986.441,E2 -17986.441} C_VEL
LIN {X 0,Y 267.248,Z 385.681,A -85,B 0,C 180,E1 -17987.225,E2 -17987.225} C_VEL
LIN {X 0,Y 263.874,Z 394.017,A -85,B 0,C 180,E1 -17988.169,E2 -17988.169} C_VEL
LIN {X 0,Y 262.95,Z 398.983,A -85,B 0,C 180,E1 -17988.848,E2 -17988.848} C_VEL
LIN {X 0,Y 262.441,Z 408.774,A -85,B 0,C 180,E1 -17990.37,E2 -17990.37} C_VEL
LIN {X 0,Y 262.044,Z 416.646,A -85,B 0,C 180,E1 -17991.911,E2 -17991.911} C_VEL
LIN {X 0,Y 261.725,Z 423.328,A -85,B 0,C 180,E1 -17993.491,E2 -17993.491} C_VEL
LIN {X 0,Y 261.526,Z 428.443,A -85,B 0,C 180,E1 -17994.926,E2 -17994.926} C_VEL
LIN {X 0,Y 261.42,Z 433.251,A -85,B 0,C 180,E1 -17996.537,E2 -17996.537} C_VEL
LIN {X 0,Y 261.212,Z 437.878,A -85,B 0,C 180,E1 -17998.463,E2 -17998.463} C_VEL
LIN {X 0,Y 261.2,Z 440.838,A -85,B 0,C 180,E1 -18000.005,E2 -18000.005} C_VEL
LIN {X 0,Y 261.308,Z 443.183,A -85,B 0,C 180,E1 -18001.546,E2 -18001.546} C_VEL
LIN {X 0,Y 261.565,Z 444.97,A -85,B 0,C 180,E1 -18003.085,E2 -18003.085} C_VEL
LIN {X 0,Y 261.995,Z 446.154,A -85,B 0,C 180,E1 -18004.621,E2 -18004.621} C_VEL
LIN {X 0,Y 262.5,Z 446.799,A -85,B 0,C 180,E1 -18006.153,E2 -18006.153} C_VEL
LIN {X 0,Y 263.023,Z 446.96,A -85,B 0,C 180,E1 -18007.682,E2 -18007.682} C_VEL
LIN {X 0,Y 263.691,Z 446.642,A -85,B 0,C 180,E1 -18009.207,E2 -18009.207} C_VEL
LIN {X 0,Y 264.906,Z 445.779,A -85,B 0,C 180,E1 -18010.707,E2 -18010.707} C_VEL
LIN {X 0,Y 266.663,Z 443.42,A -85,B 0,C 180,E1 -18012.95,E2 -18012.95} C_VEL
LIN {X 0,Y 268.887,Z 439.775,A -85,B 0,C 180,E1 -18015.156,E2 -18015.156} C_VEL
LIN {X 0,Y 271.586,Z 434.796,A -85,B 0,C 180,E1 -18017.317,E2 -18017.317} C_VEL
LIN {X 0,Y 274.627,Z 428.145,A -85,B 0,C 180,E1 -18019.436,E2 -18019.436} C_VEL
LIN {X 0,Y 276.863,Z 422.623,A -85,B 0,C 180,E1 -18020.821,E2 -18020.821} C_VEL
LIN {X 0,Y 279.897,Z 414.186,A -85,B 0,C 180,E1 -18022.519,E2 -18022.519} C_VEL
LIN {X 0,Y 282.839,Z 404.835,A -85,B 0,C 180,E1 -18024.014,E2 -18024.014} C_VEL
LIN {X 0,Y 285.243,Z 395.659,A -85,B 0,C 180,E1 -18025.156,E2 -18025.156} C_VEL
LIN {X 0,Y 287.448,Z 385.875,A -85,B 0,C 180,E1 -18026.114,E2 -18026.114} C_VEL
LIN {X 0,Y 289.613,Z 373.521,A -85,B 0,C 180,E1 -18027.02,E2 -18027.02} C_VEL
LIN {X 0,Y 291.639,Z 359.138,A -85,B 0,C 180,E1 -18027.729,E2 -18027.729} C_VEL
LIN {X 0,Y 294.576,Z 335.757,A -85,B 0,C 180,E1 -18028.809,E2 -18028.809} C_VEL
LIN {X 0,Y 291.66,Z 329.532,A -85,B 0,C 180,E1 -18030.232,E2 -18030.232} C_VEL
LIN {X 0,Y 288.584,Z 323.64,A -85,B 0,C 180,E1 -18031.884,E2 -18031.884} C_VEL
LIN {X 0,Y 285.999,Z 319.362,A -85,B 0,C 180,E1 -18033.41,E2 -18033.41} C_VEL
LIN {X 0,Y 283.684,Z 315.625,A -85,B 0,C 180,E1 -18035.002,E2 -18035.002} C_VEL
LIN {X 0,Y 280.888,Z 311.577,A -85,B 0,C 180,E1 -18037.404,E2 -18037.404} C_VEL
LIN {X 0,Y 278.42,Z 308.336,A -85,B 0,C 180,E1 -18040.51,E2 -18040.51} C_VEL
LIN {X 0,Y 277.342,Z 307.211,A -85,B 0,C 180,E1 -18043.177,E2 -18043.177} C_VEL
LIN {X 0,Y 277.435,Z 307.476,A -85,B 0,C 180,E1 -18046.541,E2 -18046.541} C_VEL
LIN {X 0,Y 278.56,Z 308.777,A -85,B 0,C 180,E1 -18049.064,E2 -18049.064} C_VEL
LIN {X 0,Y 281.929,Z 314.08,A -85,B 0,C 180,E1 -18052.997,E2 -18052.997} C_VEL
LIN {X 0,Y 284.479,Z 317.887,A -85,B 0,C 180,E1 -18054.952,E2 -18054.952} C_VEL
LIN {X 0,Y 287.795,Z 323.337,A -85,B 0,C 180,E1 -18057.042,E2 -18057.042} C_VEL
LIN {X 0,Y 290.422,Z 328.027,A -85,B 0,C 180,E1 -18058.484,E2 -18058.484} C_VEL
LIN {X 0,Y 291.082,Z 331.886,A -85,B 0,C 180,E1 -18059.066,E2 -18059.066} C_VEL
LIN {X 0,Y 291.698,Z 342.2,A -85,B 0,C 180,E1 -18060.176,E2 -18060.176} C_VEL
LIN {X 0,Y 291.981,Z 357.228,A -85,B 0,C 180,E1 -18061.499,E2 -18061.499} C_VEL
LIN {X 0,Y 291.676,Z 361.361,A -85,B 0,C 180,E1 -18061.743,E2 -18061.743} C_VEL
LIN {X 0,Y 288.027,Z 389.174,A -85,B 0,C 180,E1 -18063.068,E2 -18063.068} C_VEL
LIN {X 0,Y 285.521,Z 401.636,A -85,B 0,C 180,E1 -18063.897,E2 -18063.897} C_VEL
LIN {X 0,Y 282.923,Z 412.102,A -85,B 0,C 180,E1 -18064.824,E2 -18064.824} C_VEL
LIN {X 0,Y 279.722,Z 422.863,A -85,B 0,C 180,E1 -18066.1,E2 -18066.1} C_VEL
LIN {X 0,Y 276.875,Z 431.482,A -85,B 0,C 180,E1 -18067.423,E2 -18067.423} C_VEL
LIN {X 0,Y 273.946,Z 439.577,A -85,B 0,C 180,E1 -18068.951,E2 -18068.951} C_VEL
LIN {X 0,Y 271.077,Z 446.81,A -85,B 0,C 180,E1 -18070.697,E2 -18070.697} C_VEL
LIN {X 0,Y 268.131,Z 453.615,A -85,B 0,C 180,E1 -18072.85,E2 -18072.85} C_VEL
LIN {X 0,Y 266.042,Z 458.136,A -85,B 0,C 180,E1 -18074.682,E2 -18074.682} C_VEL
LIN {X 0,Y 264.142,Z 462.274,A -85,B 0,C 180,E1 -18076.929,E2 -18076.929} C_VEL
LIN {X 0,Y 262.708,Z 465.123,A -85,B 0,C 180,E1 -18079.206,E2 -18079.206} C_VEL
LIN {X 0,Y 262.008,Z 466.33,A -85,B 0,C 180,E1 -18080.738,E2 -18080.738} C_VEL
LIN {X 0,Y 261.539,Z 466.994,A -85,B 0,C 180,E1 -18082.278,E2 -18082.278} C_VEL
LIN {X 0,Y 261.229,Z 467.127,A -85,B 0,C 180,E1 -18084.551,E2 -18084.551} C_VEL
LIN {X 0,Y 261.27,Z 466.392,A -85,B 0,C 180,E1 -18086.626,E2 -18086.626} C_VEL
LIN {X 0,Y 261.238,Z 468.342,A -85,B 0,C 180,E1 -18088.458,E2 -18088.458} C_VEL
LIN {X 0,Y 261.252,Z 469.354,A -85,B 0,C 180,E1 -18090,E2 -18090} C_VEL
LIN {X 0,Y 261.197,Z 469.881,A -85,B 0,C 180,E1 -18091.542,E2 -18091.542} C_VEL
LIN {X 0,Y 261.185,Z 469.947,A -85,B 0,C 180,E1 -18093.085,E2 -18093.085} C_VEL
LIN {X 0,Y 261.179,Z 469.098,A -85,B 0,C 180,E1 -18095.332,E2 -18095.332} C_VEL
LIN {X 0,Y 261.503,Z 467.05,A -85,B 0,C 180,E1 -18097.722,E2 -18097.722} C_VEL
LIN {X 0,Y 262.193,Z 463.891,A -85,B 0,C 180,E1 -18100.034,E2 -18100.034} C_VEL
LIN {X 0,Y 263.293,Z 459.422,A -85,B 0,C 180,E1 -18102.33,E2 -18102.33} C_VEL
LIN {X 0,Y 264.565,Z 454.484,A -85,B 0,C 180,E1 -18104.224,E2 -18104.224} C_VEL
LIN {X 0,Y 266.066,Z 448.281,A -85,B 0,C 180,E1 -18106.102,E2 -18106.102} C_VEL
LIN {X 0,Y 267.588,Z 442.244,A -85,B 0,C 180,E1 -18107.58,E2 -18107.58} C_VEL
LIN {X 0,Y 269.326,Z 434.918,A -85,B 0,C 180,E1 -18109.037,E2 -18109.037} C_VEL
LIN {X 0,Y 270.383,Z 429.56,A -85,B 0,C 180,E1 -18109.947,E2 -18109.947} C_VEL
LIN {X 0,Y 271.999,Z 421.852,A -85,B 0,C 180,E1 -18111.008,E2 -18111.008} C_VEL
LIN {X 0,Y 273.257,Z 414.024,A -85,B 0,C 180,E1 -18111.896,E2 -18111.896} C_VEL
LIN {X 0,Y 274.71,Z 404.114,A -85,B 0,C 180,E1 -18112.743,E2 -18112.743} C_VEL
LIN {X 0,Y 275.823,Z 394.721,A -85,B 0,C 180,E1 -18113.321,E2 -18113.321} C_VEL
LIN {X 0,Y 276.508,Z 385.052,A -85,B 0,C 180,E1 -18113.73,E2 -18113.73} C_VEL
LIN {X 0,Y 277.399,Z 354.186,A -85,B 0,C 180,E1 -18114.576,E2 -18114.576} C_VEL
LIN {X 0,Y 275.316,Z 339.945,A -85,B 0,C 180,E1 -18115.253,E2 -18115.253} C_VEL
LIN {X 0,Y 271.754,Z 321.607,A -85,B 0,C 180,E1 -18116.263,E2 -18116.263} C_VEL
LIN {X 0,Y 269.579,Z 312.794,A -85,B 0,C 180,E1 -18116.822,E2 -18116.822} C_VEL
LIN {X 0,Y 267.719,Z 308.066,A -85,B 0,C 180,E1 -18117.237,E2 -18117.237} C_VEL
LIN {X 0,Y 265.821,Z 298.734,A -85,B 0,C 180,E1 -18121.034,E2 -18121.034} C_VEL
LIN {X 0,Y 263.676,Z 289.622,A -85,B 0,C 180,E1 -18125.017,E2 -18125.017} C_VEL
LIN {X 0,Y 263.21,Z 287.498,A -85,B 0,C 180,E1 -18126.071,E2 -18126.071} C_VEL
LIN {X 0,Y 263.116,Z 287.523,A -85,B 0,C 180,E1 -18129.87,E2 -18129.87} C_VEL
LIN {X 0,Y 263.113,Z 287.518,A -85,B 0,C 180,E1 -18133.986,E2 -18133.986} C_VEL
LIN {X 0,Y 263.085,Z 287.523,A -85,B 0,C 180,E1 -18138.094,E2 -18138.094} C_VEL
LIN {X 0,Y 263.123,Z 287.52,A -85,B 0,C 180,E1 -18142.092,E2 -18142.092} C_VEL
LIN {X 0,Y 263.16,Z 287.512,A -85,B 0,C 180,E1 -18145.882,E2 -18145.882} C_VEL
LIN {X 0,Y 263.134,Z 287.511,A -85,B 0,C 180,E1 -18149.5,E2 -18149.5} C_VEL
LIN {X 0,Y 263.152,Z 287.511,A -85,B 0,C 180,E1 -18152.994,E2 -18152.994} C_VEL
LIN {X 0,Y 263.155,Z 287.517,A -85,B 0,C 180,E1 -18156.38,E2 -18156.38} C_VEL
LIN {X 0,Y 263.249,Z 287.497,A -85,B 0,C 180,E1 -18159.688,E2 -18159.688} C_VEL
LIN {X 0,Y 263.328,Z 287.485,A -85,B 0,C 180,E1 -18164.516,E2 -18164.516} C_VEL
LIN {X 0,Y 263.359,Z 287.474,A -85,B 0,C 180,E1 -18169.229,E2 -18169.229} C_VEL
LIN {X 0,Y 263.561,Z 287.46,A -85,B 0,C 180,E1 -18172.333,E2 -18172.333} C_VEL
LIN {X 0,Y 263.747,Z 287.433,A -85,B 0,C 180,E1 -18178.468,E2 -18178.468} C_VEL
LIN {X 0,Y 263.748,Z 287.435,A -85,B 0,C 180,E1 -18181.522,E2 -18181.522} C_VEL
LIN {X 0,Y 263.529,Z 287.468,A -85,B 0,C 180,E1 -18187.658,E2 -18187.658} C_VEL
LIN {X 0,Y 263.348,Z 287.481,A -85,B 0,C 180,E1 -18190.761,E2 -18190.761} C_VEL
LIN {X 0,Y 263.344,Z 287.483,A -85,B 0,C 180,E1 -18195.473,E2 -18195.473} C_VEL
LIN {X 0,Y 263.255,Z 287.496,A -85,B 0,C 180,E1 -18200.301,E2 -18200.301} C_VEL
LIN {X 0,Y 263.197,Z 287.507,A -85,B 0,C 180,E1 -18205.286,E2 -18205.286} C_VEL
LIN {X 0,Y 263.152,Z 287.513,A -85,B 0,C 180,E1 -18208.726,E2 -18208.726} C_VEL
LIN {X 0,Y 263.117,Z 287.519,A -85,B 0,C 180,E1 -18212.283,E2 -18212.283} C_VEL
LIN {X 0,Y 263.178,Z 287.501,A -85,B 0,C 180,E1 -18216.762,E2 -18216.762} C_VEL
LIN {X 0,Y 263.186,Z 287.51,A -85,B 0,C 180,E1 -18221.609,E2 -18221.609} C_VEL
LIN {X 0,Y 263.207,Z 287.641,A -85,B 0,C 180,E1 -18225.098,E2 -18225.098} C_VEL
LIN {X 0,Y 264.433,Z 290.715,A -85,B 0,C 180,E1 -18225.433,E2 -18225.433} C_VEL
LIN {X 0,Y 265.908,Z 293.153,A -85,B 0,C 180,E1 -18225.724,E2 -18225.724} C_VEL
LIN {X 0,Y 270.828,Z 302.635,A -85,B 0,C 180,E1 -18226.7,E2 -18226.7} C_VEL
LIN {X 0,Y 277.45,Z 317.439,A -85,B 0,C 180,E1 -18228.004,E2 -18228.004} C_VEL
LIN {X 0,Y 278.554,Z 320.133,A -85,B 0,C 180,E1 -18228.22,E2 -18228.22} C_VEL
LIN {X 0,Y 277.064,Z 364.46,A -85,B 0,C 180,E1 -18229.42,E2 -18229.42} C_VEL
LIN {X 0,Y 276.425,Z 374.583,A -85,B 0,C 180,E1 -18229.905,E2 -18229.905} C_VEL
LIN {X 0,Y 275.229,Z 386.719,A -85,B 0,C 180,E1 -18230.803,E2 -18230.803} C_VEL
LIN {X 0,Y 273.896,Z 395.98,A -85,B 0,C 180,E1 -18231.755,E2 -18231.755} C_VEL
LIN {X 0,Y 272.555,Z 404.214,A -85,B 0,C 180,E1 -18232.84,E2 -18232.84} C_VEL
LIN {X 0,Y 271.068,Z 411.855,A -85,B 0,C 180,E1 -18234.084,E2 -18234.084} C_VEL
LIN {X 0,Y 269.505,Z 418.704,A -85,B 0,C 180,E1 -18235.446,E2 -18235.446} C_VEL
LIN {X 0,Y 267.89,Z 425.341,A -85,B 0,C 180,E1 -18237.076,E2 -18237.076} C_VEL
LIN {X 0,Y 266.216,Z 431.657,A -85,B 0,C 180,E1 -18239.017,E2 -18239.017} C_VEL
LIN {X 0,Y 264.537,Z 437.467,A -85,B 0,C 180,E1 -18241.432,E2 -18241.432} C_VEL
LIN {X 0,Y 263.23,Z 441.652,A -85,B 0,C 180,E1 -18243.862,E2 -18243.862} C_VEL
LIN {X 0,Y 262.234,Z 444.457,A -85,B 0,C 180,E1 -18246.297,E2 -18246.297} C_VEL
LIN {X 0,Y 261.755,Z 445.513,A -85,B 0,C 180,E1 -18247.921,E2 -18247.921} C_VEL
LIN {X 0,Y 261.302,Z 446.165,A -85,B 0,C 180,E1 -18250.261,E2 -18250.261} C_VEL
LIN {X 0,Y 261.046,Z 445.528,A -85,B 0,C 180,E1 -18252.774,E2 -18252.774} C_VEL
LIN {X 0,Y 261.06,Z 444.475,A -85,B 0,C 180,E1 -18254.383,E2 -18254.383} C_VEL
LIN {X 0,Y 261.272,Z 441.748,A -85,B 0,C 180,E1 -18256.783,E2 -18256.783} C_VEL
LIN {X 0,Y 261.536,Z 439.269,A -85,B 0,C 180,E1 -18258.373,E2 -18258.373} C_VEL
LIN {X 0,Y 261.842,Z 436.124,A -85,B 0,C 180,E1 -18259.953,E2 -18259.953} C_VEL
LIN {X 0,Y 262.543,Z 429.96,A -85,B 0,C 180,E1 -18262.308,E2 -18262.308} C_VEL
LIN {X 0,Y 262.983,Z 424.879,A -85,B 0,C 180,E1 -18263.864,E2 -18263.864} C_VEL
LIN {X 0,Y 263.709,Z 418.704,A -85,B 0,C 180,E1 -18265.415,E2 -18265.415} C_VEL
LIN {X 0,Y 264.525,Z 411.194,A -85,B 0,C 180,E1 -18266.954,E2 -18266.954} C_VEL
LIN {X 0,Y 265.37,Z 403.138,A -85,B 0,C 180,E1 -18268.293,E2 -18268.293} C_VEL
LIN {X 0,Y 266.326,Z 393.051,A -85,B 0,C 180,E1 -18269.622,E2 -18269.622} C_VEL
LIN {X 0,Y 267.094,Z 382.098,A -85,B 0,C 180,E1 -18270.674,E2 -18270.674} C_VEL
LIN {X 0,Y 267.592,Z 372.674,A -85,B 0,C 180,E1 -18271.332,E2 -18271.332} C_VEL
LIN {X 0,Y 267.9,Z 363.133,A -85,B 0,C 180,E1 -18271.788,E2 -18271.788} C_VEL
LIN {X 0,Y 268.977,Z 311.219,A -85,B 0,C 180,E1 -18273.207,E2 -18273.207} C_VEL
LIN {X 0,Y 266.757,Z 297.697,A -85,B 0,C 180,E1 -18273.715,E2 -18273.715} C_VEL
LIN {X 0,Y 263.364,Z 287.493,A -85,B 0,C 180,E1 -18274.257,E2 -18274.257} C_VEL
LIN {X 0,Y 263.526,Z 287.47,A -85,B 0,C 180,E1 -18277.663,E2 -18277.663} C_VEL
LIN {X 0,Y 263.32,Z 287.497,A -85,B 0,C 180,E1 -18280.768,E2 -18280.768} C_VEL
LIN {X 0,Y 263.298,Z 287.5,A -85,B 0,C 180,E1 -18285.481,E2 -18285.481} C_VEL
LIN {X 0,Y 263.234,Z 287.505,A -85,B 0,C 180,E1 -18290.309,E2 -18290.309} C_VEL
LIN {X 0,Y 263.14,Z 287.521,A -85,B 0,C 180,E1 -18295.299,E2 -18295.299} C_VEL
LIN {X 0,Y 263.103,Z 287.522,A -85,B 0,C 180,E1 -18298.739,E2 -18298.739} C_VEL
LIN {X 0,Y 263.102,Z 287.518,A -85,B 0,C 180,E1 -18302.293,E2 -18302.293} C_VEL
LIN {X 0,Y 263.15,Z 287.515,A -85,B 0,C 180,E1 -18306.765,E2 -18306.765} C_VEL
LIN {X 0,Y 263.068,Z 287.528,A -85,B 0,C 180,E1 -18309.88,E2 -18309.88} C_VEL
LIN {X 0,Y 263.077,Z 287.526,A -85,B 0,C 180,E1 -18313.994,E2 -18313.994} C_VEL
LIN {X 0,Y 263.106,Z 287.521,A -85,B 0,C 180,E1 -18318.412,E2 -18318.412} C_VEL
LIN {X 0,Y 263.169,Z 287.514,A -85,B 0,C 180,E1 -18323.241,E2 -18323.241} C_VEL
LIN {X 0,Y 263.115,Z 287.522,A -85,B 0,C 180,E1 -18327.716,E2 -18327.716} C_VEL
LIN {X 0,Y 263.137,Z 287.521,A -85,B 0,C 180,E1 -18331.81,E2 -18331.81} C_VEL
LIN {X 0,Y 263.181,Z 287.51,A -85,B 0,C 180,E1 -18335.223,E2 -18335.223} C_VEL
LIN {X 0,Y 263.26,Z 287.493,A -85,B 0,C 180,E1 -18339.699,E2 -18339.699} C_VEL
LIN {X 0,Y 263.419,Z 287.46,A -85,B 0,C 180,E1 -18342.239,E2 -18342.239} C_VEL
LIN {X 0,Y 265.683,Z 308.619,A -85,B 0,C 180,E1 -18343.194,E2 -18343.194} C_VEL
LIN {X 0,Y 264.338,Z 365.045,A -85,B 0,C 180,E1 -18345.67,E2 -18345.67} C_VEL
LIN {X 0,Y 263.957,Z 376.549,A -85,B 0,C 180,E1 -18346.435,E2 -18346.435} C_VEL
LIN {X 0,Y 263.516,Z 388.049,A -85,B 0,C 180,E1 -18347.491,E2 -18347.491} C_VEL
LIN {X 0,Y 263.042,Z 397.486,A -85,B 0,C 180,E1 -18348.641,E2 -18348.641} C_VEL
LIN {X 0,Y 262.95,Z 398.983,A -85,B 0,C 180,E1 -18348.848,E2 -18348.848} C_VEL
LIN {X 0,Y 261.982,Z 403.829,A -85,B 0,C 180,E1 -18349.565,E2 -18349.565} C_VEL
LIN {X 0,Y 258.714,Z 411.045,A -85,B 0,C 180,E1 -18350.871,E2 -18350.871} C_VEL
